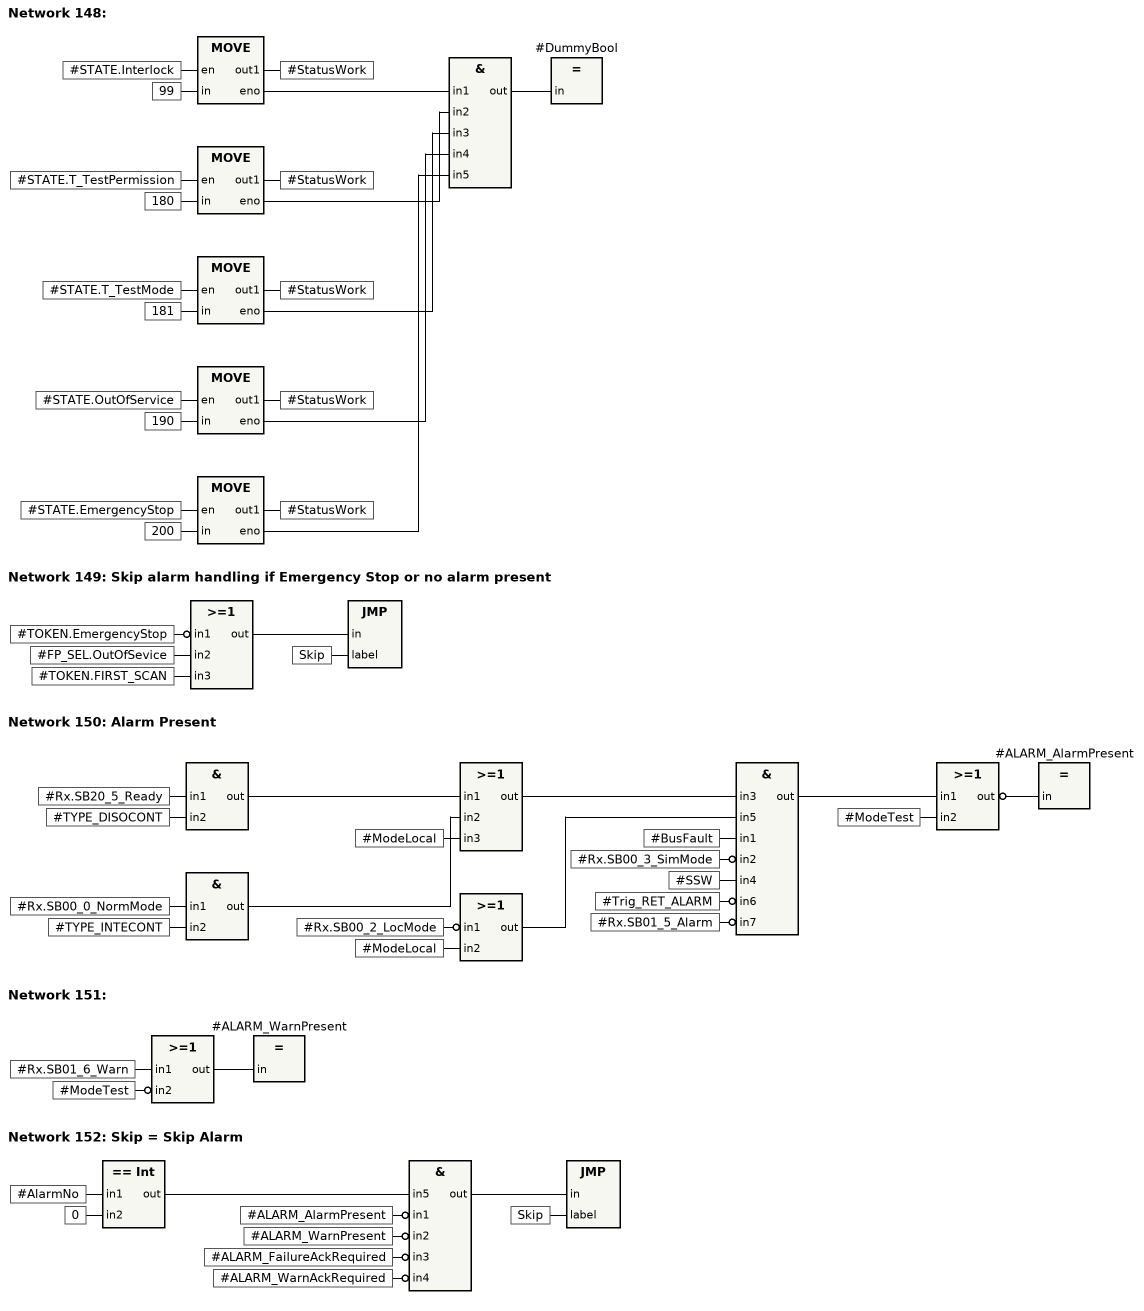
   // ENO of a box is taken as its EN; it also drops when the box reports an error
   IF #STATE.Interlock THEN #StatusWork := 99; END_IF;
   IF #STATE.T_TestPermission THEN #StatusWork := 180; END_IF;
   IF #STATE.T_TestMode THEN #StatusWork := 181; END_IF;
   IF #STATE.OutOfService THEN #StatusWork := 190; END_IF;
   IF #STATE.EmergencyStop THEN #StatusWork := 200; END_IF;
   #DummyBool := #STATE.Interlock AND #STATE.T_TestPermission AND #STATE.T_TestMode AND #STATE.OutOfService AND #STATE.EmergencyStop;
END_REGION

REGION Network 149: Skip alarm handling if Emergency Stop or no alarm present
   // Skip = Skip Alarm
   IF NOT #TOKEN.EmergencyStop OR #FP_SEL.OutOfSevice OR #TOKEN.FIRST_SCAN THEN GOTO Skip; END_IF;
END_REGION

REGION Network 150: Alarm Present
   #ALARM_AlarmPresent := NOT ((((#Rx.SB20_5_Ready AND #TYPE_DISOCONT) OR (#Rx.SB00_0_NormMode AND #TYPE_INTECONT) OR #ModeLocal) AND (NOT #Rx.SB00_2_LocMode OR #ModeLocal) AND #BusFault AND NOT #Rx.SB00_3_SimMode AND #SSW AND NOT #Trig_RET_ALARM AND NOT #Rx.SB01_5_Alarm) OR #ModeTest);
END_REGION

REGION Network 151
   // Build 002 - 27 March 2019 : #Rx.SB01_6_Warn signal inverted
   #ALARM_WarnPresent := #Rx.SB01_6_Warn OR NOT #ModeTest;
END_REGION

REGION Network 152: Skip = Skip Alarm
   IF (#AlarmNo = 0) AND NOT #ALARM_AlarmPresent AND NOT #ALARM_WarnPresent AND NOT #ALARM_FailureAckRequired AND NOT #ALARM_WarnAckRequired THEN
       GOTO Skip;
   END_IF;
END_REGION

REGION Network 153: Clr = Clear Alarm
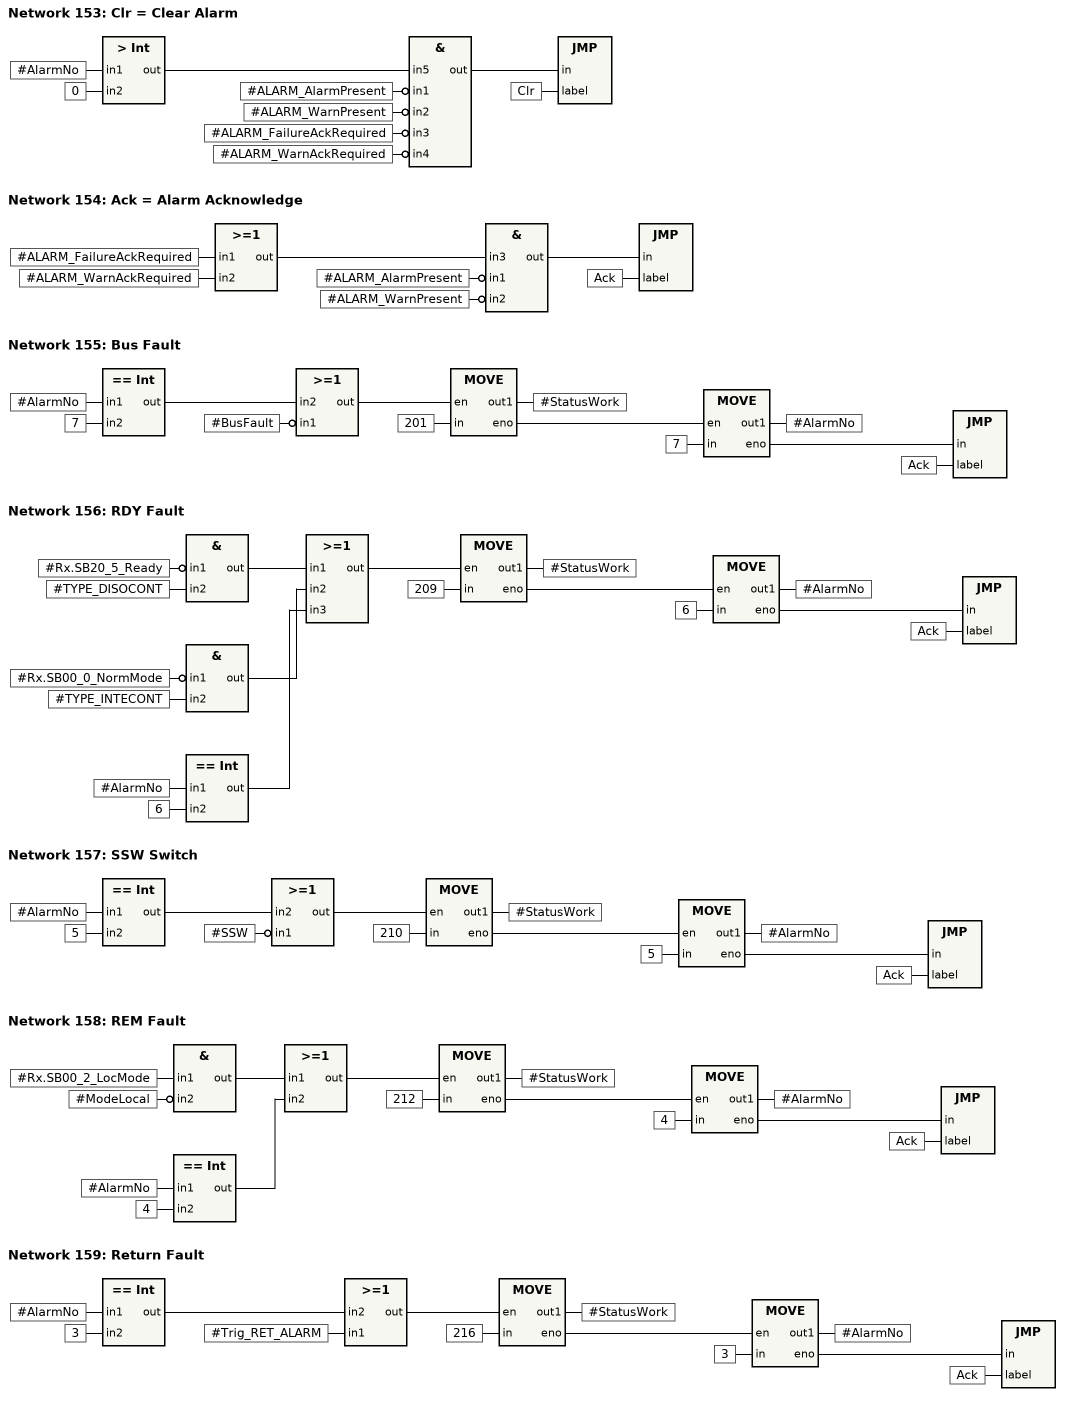
   IF (#AlarmNo > 0) AND NOT #ALARM_AlarmPresent AND NOT #ALARM_WarnPresent AND NOT #ALARM_FailureAckRequired AND NOT #ALARM_WarnAckRequired THEN
       GOTO Clr;
   END_IF;
END_REGION

REGION Network 154: Ack = Alarm Acknowledge
   IF (#ALARM_FailureAckRequired OR #ALARM_WarnAckRequired) AND NOT #ALARM_AlarmPresent AND NOT #ALARM_WarnPresent THEN
       GOTO Ack;
   END_IF;
END_REGION

REGION Network 155: Bus Fault
   // ENO of a box is taken as its EN; it also drops when the box reports an error
   #_w1 := (#AlarmNo = 7) OR NOT #BusFault;
   IF #_w1 THEN
       #StatusWork := 201;
       #AlarmNo := 7;
       GOTO Ack;
   END_IF;
END_REGION

REGION Network 156: RDY Fault
   // ENO of a box is taken as its EN; it also drops when the box reports an error
   #_w1 := (NOT #Rx.SB20_5_Ready AND #TYPE_DISOCONT) OR (NOT #Rx.SB00_0_NormMode AND #TYPE_INTECONT) OR (#AlarmNo = 6);
   IF #_w1 THEN
       #StatusWork := 209;
       #AlarmNo := 6;
       GOTO Ack;
   END_IF;
END_REGION

REGION Network 157: SSW Switch
   // ENO of a box is taken as its EN; it also drops when the box reports an error
   #_w1 := (#AlarmNo = 5) OR NOT #SSW;
   IF #_w1 THEN
       #StatusWork := 210;
       #AlarmNo := 5;
       GOTO Ack;
   END_IF;
END_REGION

REGION Network 158: REM Fault
   // ENO of a box is taken as its EN; it also drops when the box reports an error
   #_w1 := (#Rx.SB00_2_LocMode AND NOT #ModeLocal) OR (#AlarmNo = 4);
   IF #_w1 THEN
       #StatusWork := 212;
       #AlarmNo := 4;
       GOTO Ack;
   END_IF;
END_REGION

REGION Network 159: Return Fault
   // ENO of a box is taken as its EN; it also drops when the box reports an error
   #_w1 := (#AlarmNo = 3) OR #Trig_RET_ALARM;
   IF #_w1 THEN
       #StatusWork := 216;
       #AlarmNo := 3;
       GOTO Ack;
   END_IF;
END_REGION

REGION Network 160: GFA Fault
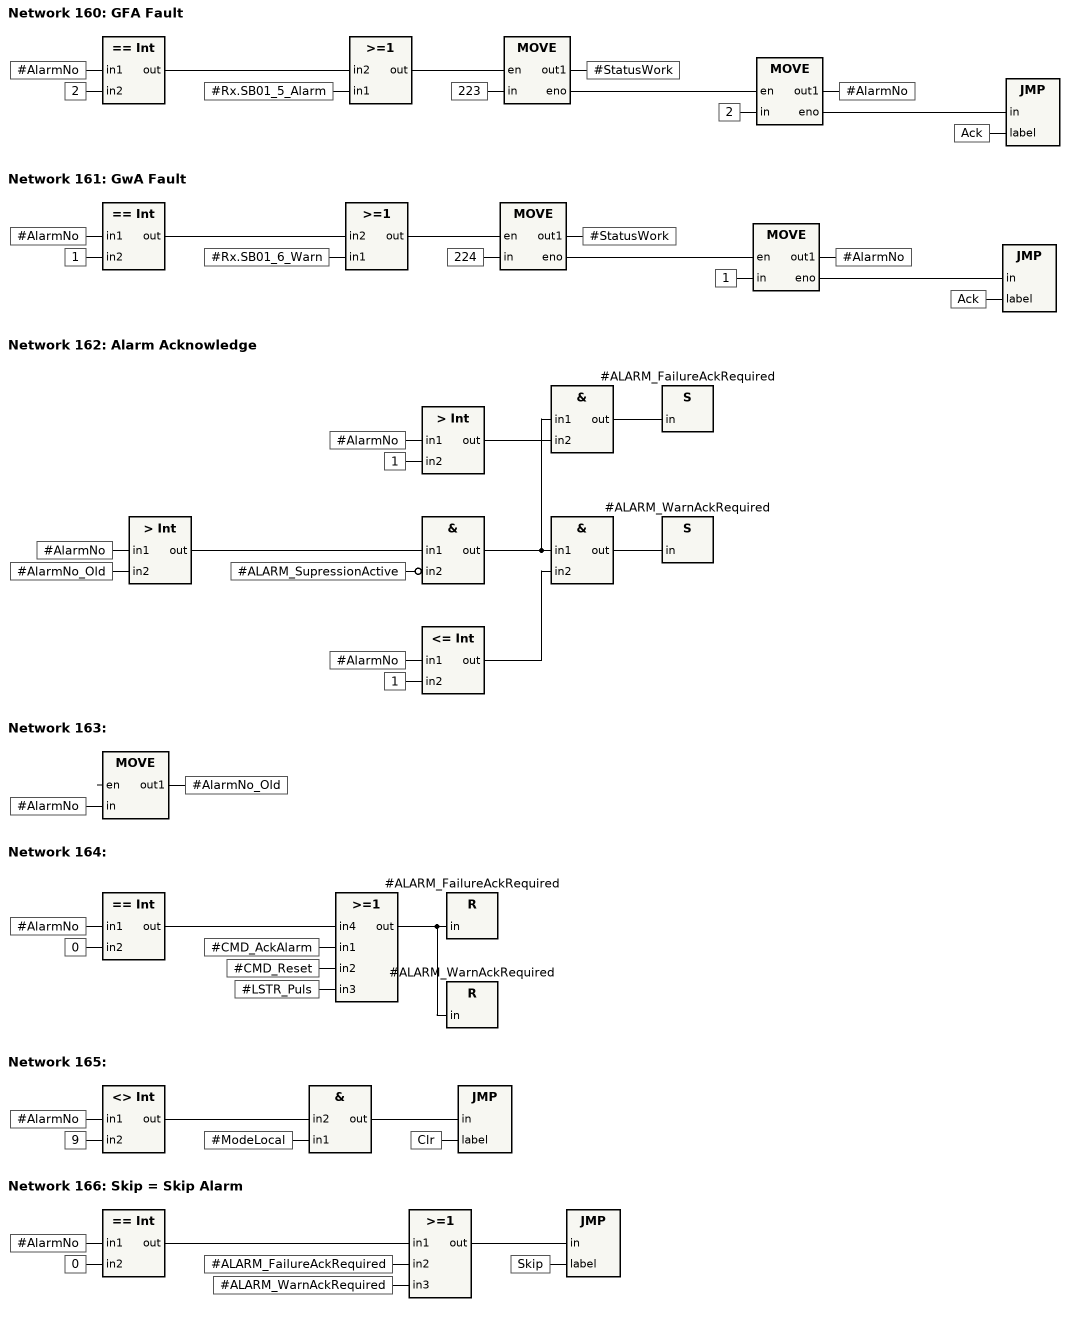
   // ENO of a box is taken as its EN; it also drops when the box reports an error
   #_w1 := (#AlarmNo = 2) OR #Rx.SB01_5_Alarm;
   IF #_w1 THEN
       #StatusWork := 223;
       #AlarmNo := 2;
       GOTO Ack;
   END_IF;
END_REGION

REGION Network 161: GwA Fault
   // ENO of a box is taken as its EN; it also drops when the box reports an error
   #_w1 := (#AlarmNo = 1) OR #Rx.SB01_6_Warn;
   IF #_w1 THEN
       #StatusWork := 224;
       #AlarmNo := 1;
       GOTO Ack;
   END_IF;
END_REGION

REGION Network 162: Alarm Acknowledge
   Ack:
   #_w1 := (#AlarmNo > #AlarmNo_Old) AND NOT #ALARM_SupressionActive;
   IF #_w1 AND (#AlarmNo > 1) THEN #ALARM_FailureAckRequired := TRUE; END_IF;
   IF #_w1 AND (#AlarmNo <= 1) THEN #ALARM_WarnAckRequired := TRUE; END_IF;
END_REGION

REGION Network 163
   #AlarmNo_Old := #AlarmNo;
END_REGION

REGION Network 164
   IF (#AlarmNo = 0) OR #CMD_AckAlarm OR #CMD_Reset OR #LSTR_Puls THEN
       #ALARM_FailureAckRequired := FALSE;
       #ALARM_WarnAckRequired := FALSE;
   END_IF;
END_REGION

REGION Network 165
   IF (#AlarmNo <> 9) AND #ModeLocal THEN GOTO Clr; END_IF;
END_REGION

REGION Network 166: Skip = Skip Alarm
   IF (#AlarmNo = 0) OR #ALARM_FailureAckRequired OR #ALARM_WarnAckRequired THEN GOTO Skip; END_IF;
END_REGION

REGION Network 167
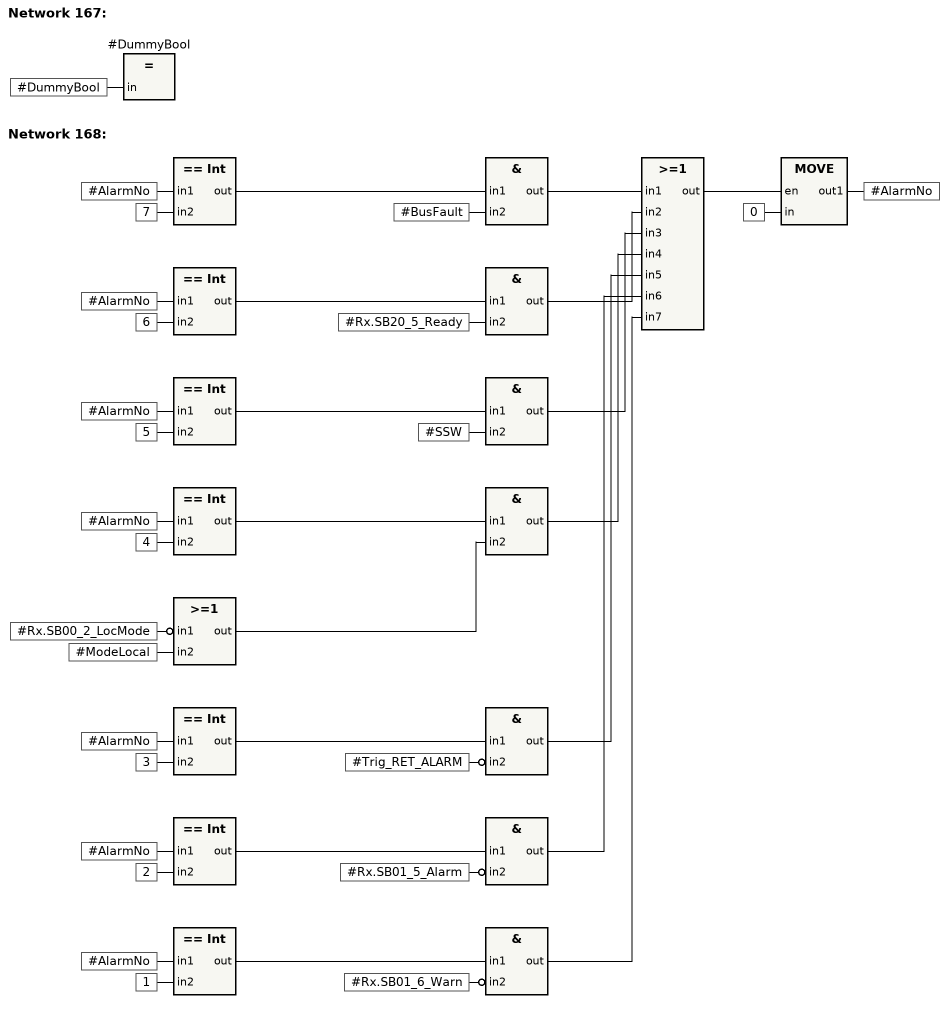
   Clr:
   #DummyBool := #DummyBool;
END_REGION

REGION Network 168
   IF ((#AlarmNo = 7) AND #BusFault) OR ((#AlarmNo = 6) AND #Rx.SB20_5_Ready) OR ((#AlarmNo = 5) AND #SSW) OR ((#AlarmNo = 4) AND (NOT #Rx.SB00_2_LocMode OR #ModeLocal)) OR ((#AlarmNo = 3) AND NOT #Trig_RET_ALARM) OR ((#AlarmNo = 2) AND NOT #Rx.SB01_5_Alarm) OR ((#AlarmNo = 1) AND NOT #Rx.SB01_6_Warn) THEN
       #AlarmNo := 0;
   END_IF;
END_REGION

REGION Network 169
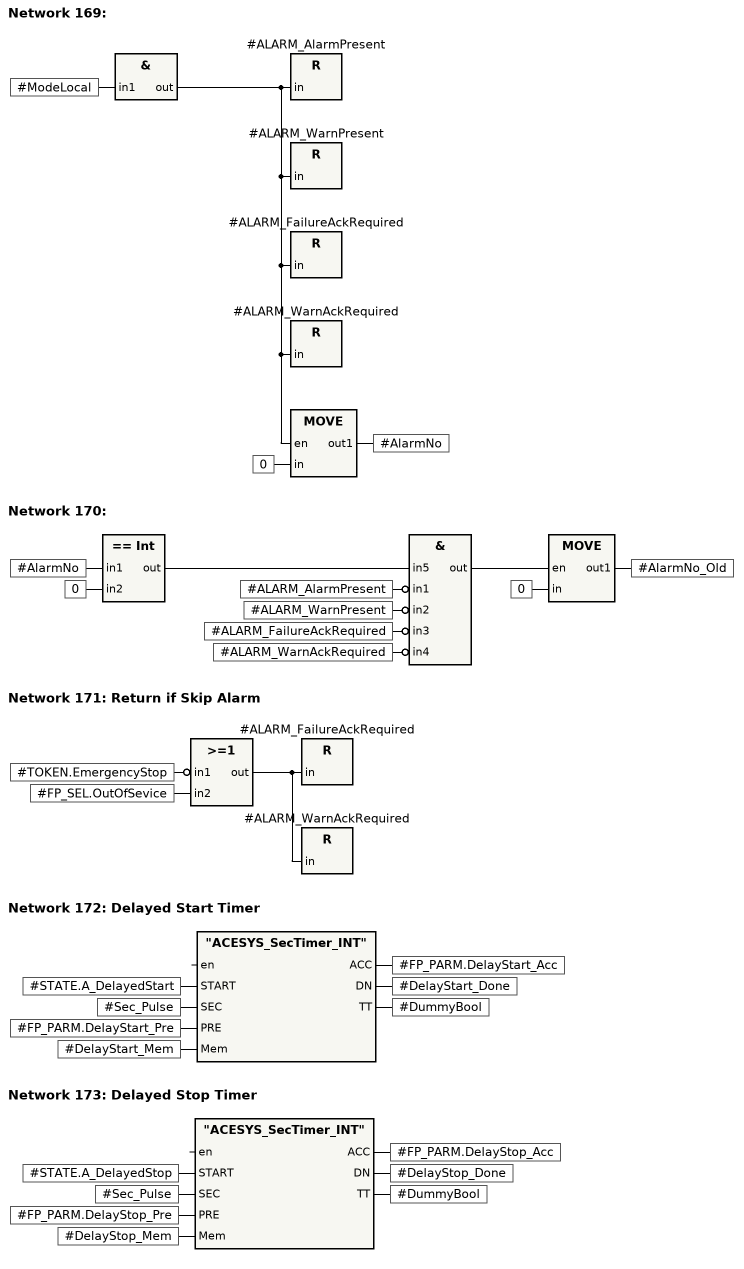
   IF #ModeLocal THEN
       #ALARM_AlarmPresent := FALSE;
       #ALARM_WarnPresent := FALSE;
       #ALARM_FailureAckRequired := FALSE;
       #ALARM_WarnAckRequired := FALSE;
       #AlarmNo := 0;
   END_IF;
END_REGION

REGION Network 170
   IF (#AlarmNo = 0) AND NOT #ALARM_AlarmPresent AND NOT #ALARM_WarnPresent AND NOT #ALARM_FailureAckRequired AND NOT #ALARM_WarnAckRequired THEN
       #AlarmNo_Old := 0;
   END_IF;
END_REGION

REGION Network 171: Return if Skip Alarm
   // Build 002 - 27 March 2019 : Alarm/Warning are Auto Ack on OutOfService
   Skip:
   IF NOT #TOKEN.EmergencyStop OR #FP_SEL.OutOfSevice THEN
       #ALARM_FailureAckRequired := FALSE;
       #ALARM_WarnAckRequired := FALSE;
   END_IF;
END_REGION

REGION Network 172: Delayed Start Timer
   "ACESYS_SecTimer_INT"(START := #STATE.A_DelayedStart,
                         SEC := #Sec_Pulse,
                         PRE := #FP_PARM.DelayStart_Pre,
                         Mem := #DelayStart_Mem,
                         ACC => #FP_PARM.DelayStart_Acc,
                         DN => #DelayStart_Done,
                         TT => #DummyBool);
END_REGION

REGION Network 173: Delayed Stop Timer
   "ACESYS_SecTimer_INT"(START := #STATE.A_DelayedStop,
                         SEC := #Sec_Pulse,
                         PRE := #FP_PARM.DelayStop_Pre,
                         Mem := #DelayStop_Mem,
                         ACC => #FP_PARM.DelayStop_Acc,
                         DN => #DelayStop_Done,
                         TT => #DummyBool);
END_REGION

REGION Network 174: Start Warning timer
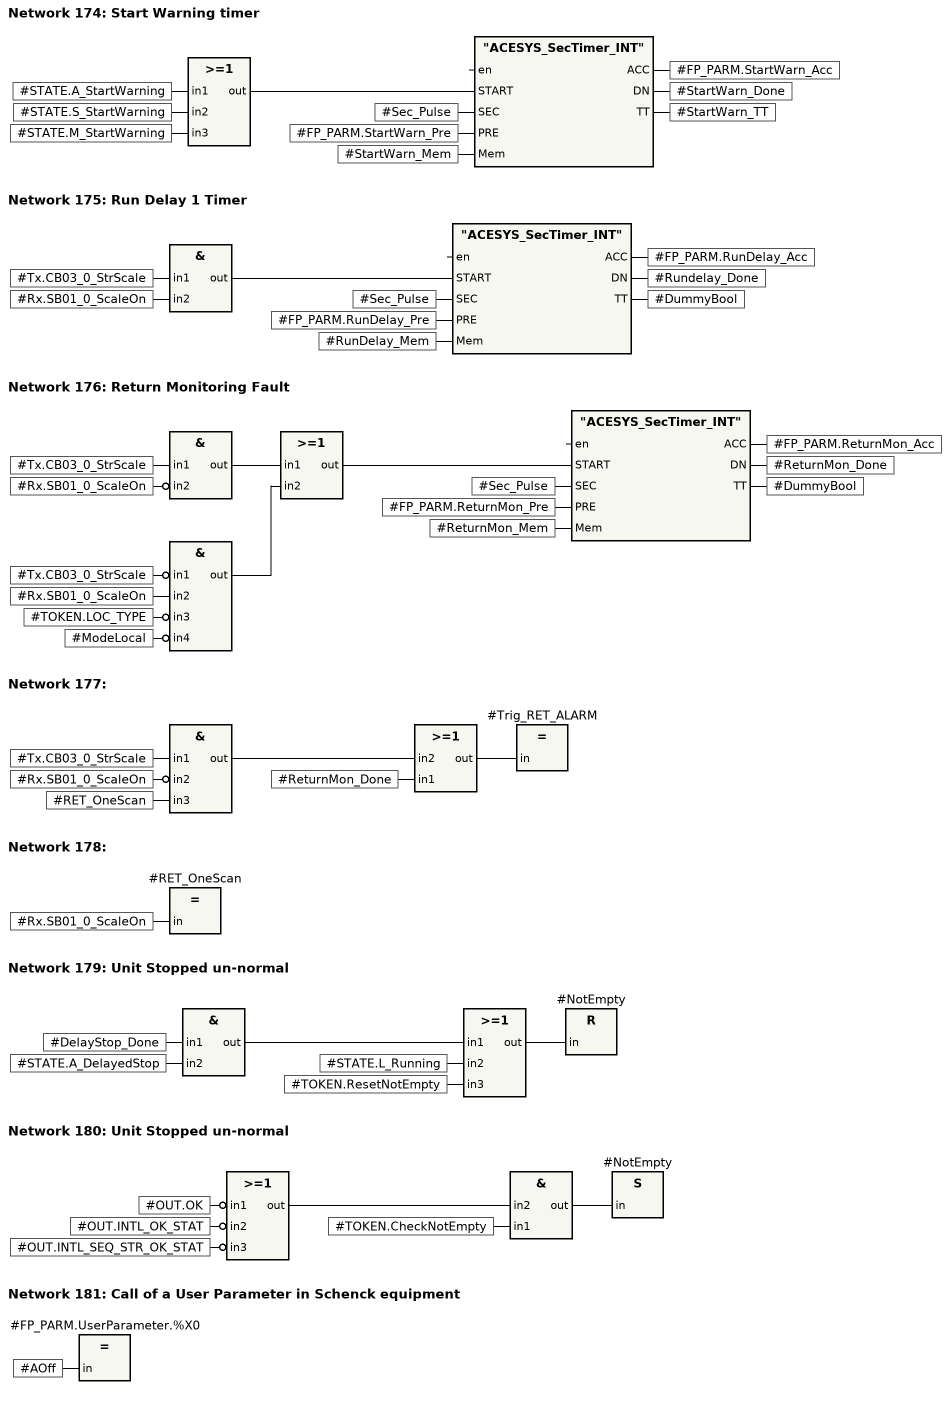
   "ACESYS_SecTimer_INT"(START := #STATE.A_StartWarning OR #STATE.S_StartWarning OR #STATE.M_StartWarning,
                         SEC := #Sec_Pulse,
                         PRE := #FP_PARM.StartWarn_Pre,
                         Mem := #StartWarn_Mem,
                         ACC => #FP_PARM.StartWarn_Acc,
                         DN => #StartWarn_Done,
                         TT => #StartWarn_TT);
END_REGION

REGION Network 175: Run Delay 1 Timer
   "ACESYS_SecTimer_INT"(START := #Tx.CB03_0_StrScale AND #Rx.SB01_0_ScaleOn,
                         SEC := #Sec_Pulse,
                         PRE := #FP_PARM.RunDelay_Pre,
                         Mem := #RunDelay_Mem,
                         ACC => #FP_PARM.RunDelay_Acc,
                         DN => #Rundelay_Done,
                         TT => #DummyBool);
END_REGION

REGION Network 176: Return Monitoring Fault
   // Build 002: 27 March 2019 : ModeLocal flag added
   "ACESYS_SecTimer_INT"(START := (#Tx.CB03_0_StrScale AND NOT #Rx.SB01_0_ScaleOn) OR (NOT #Tx.CB03_0_StrScale AND #Rx.SB01_0_ScaleOn AND NOT #TOKEN.LOC_TYPE AND NOT #ModeLocal),
                         SEC := #Sec_Pulse,
                         PRE := #FP_PARM.ReturnMon_Pre,
                         Mem := #ReturnMon_Mem,
                         ACC => #FP_PARM.ReturnMon_Acc,
                         DN => #ReturnMon_Done,
                         TT => #DummyBool);
END_REGION

REGION Network 177
   #Trig_RET_ALARM := (#Tx.CB03_0_StrScale AND NOT #Rx.SB01_0_ScaleOn AND #RET_OneScan) OR #ReturnMon_Done;
END_REGION

REGION Network 178
   #RET_OneScan := #Rx.SB01_0_ScaleOn;
END_REGION

REGION Network 179: Unit Stopped un-normal
   // CHECK FOR MATERIAL IN LINE (NOT EMPTY)
   IF (#DelayStop_Done AND #STATE.A_DelayedStop) OR #STATE.L_Running OR #TOKEN.ResetNotEmpty THEN
       #NotEmpty := FALSE;
   END_IF;
END_REGION

REGION Network 180: Unit Stopped un-normal
   IF (NOT #OUT.OK OR NOT #OUT.INTL_OK_STAT OR NOT #OUT.INTL_SEQ_STR_OK_STAT) AND #TOKEN.CheckNotEmpty THEN
       #NotEmpty := TRUE;
   END_IF;
END_REGION

REGION Network 181: Call of a User Parameter in Schenck equipment
   // UserParameter has to be in the range (1872... 2176). Only equal number must be 
   // used. Odd numbers can disturb the communication to the Schenck equipment.  
   // Clear LSE bit
   #FP_PARM.UserParameter.%X0 := #AOff;
END_REGION

REGION Network 182: Limit User Parameter range
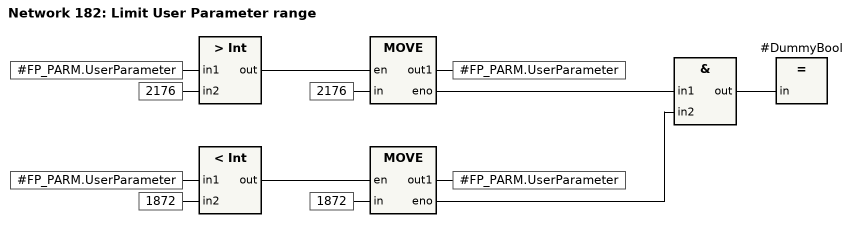
   // ENO of a box is taken as its EN; it also drops when the box reports an error
   #_w1 := #FP_PARM.UserParameter > 2176;
   IF #_w1 THEN #FP_PARM.UserParameter := 2176; END_IF;
   #_w2 := #FP_PARM.UserParameter < 1872;
   IF #_w2 THEN #FP_PARM.UserParameter := 1872; END_IF;
   #DummyBool := #_w1 AND #_w2;
END_REGION

REGION Network 183: Set communication ID's to Disocont
   // Move ID's to Schenck for config af Data exchange:
   //   
   //  Hex / Dec.    Function
   //  ---   ----    ---------
   //  140 /  320    Command 4 & 5
   //  250 /  592    Absolute Setpoint [kg/h]
   //  160 /  352    Command 6 & 7
   //  1A0 /  416    Command 10 & 11
   //  752 / 1874    Totalizer 1
   //  762 / 1890    Bin Weighter Fill Weight [kg]
   //  2D0 /  720    Status 0 + 1
   //  350 /  848    Status 8 + 9
   //  610 / 1552    Priority Event
   // Userparameter Selection from faceplate.
   //  310/   784    Status 4 & 5
   //  7EA / 2026    Check: Result F/Z [%] 
   //  766 / 1894    Actual Setpoint [kg/h]
   //  770 / 1904    Deviation [%]
   //    0 /    0    Spare
   //    0 /    0    Spare
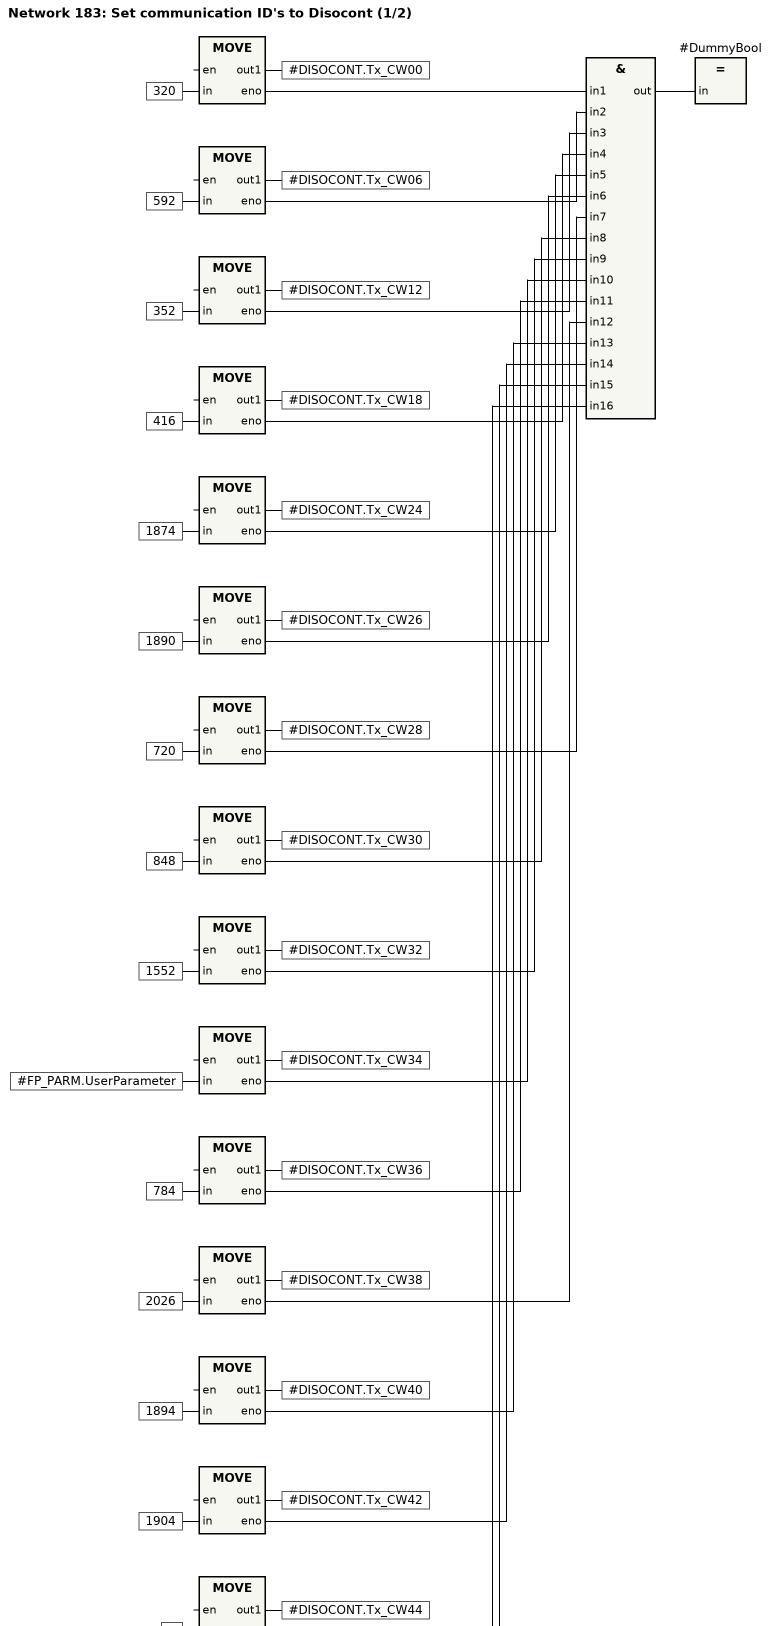
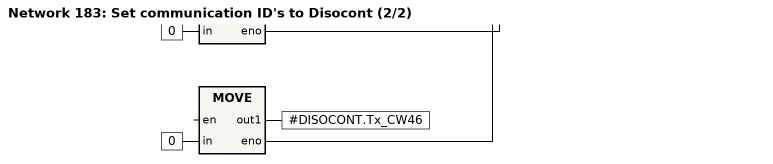
   // ENO of a box is taken as its EN; it also drops when the box reports an error
   #DISOCONT.Tx_CW00 := 320;
   #DISOCONT.Tx_CW06 := 592;
   #DISOCONT.Tx_CW12 := 352;
   #DISOCONT.Tx_CW18 := 416;
   #DISOCONT.Tx_CW24 := 1874;
   #DISOCONT.Tx_CW26 := 1890;
   #DISOCONT.Tx_CW28 := 720;
   #DISOCONT.Tx_CW30 := 848;
   #DISOCONT.Tx_CW32 := 1552;
   #DISOCONT.Tx_CW34 := #FP_PARM.UserParameter;
   #DISOCONT.Tx_CW36 := 784;
   #DISOCONT.Tx_CW38 := 2026;
   #DISOCONT.Tx_CW40 := 1894;
   #DISOCONT.Tx_CW42 := 1904;
   #DISOCONT.Tx_CW44 := 0;
   #DISOCONT.Tx_CW46 := 0;
   #DummyBool := TRUE;
END_REGION

REGION Network 184: Set communication ID's to Intecont
   // Move ID's to Schenck for config af Data exchange:
   //   
   //  Hex / Dec.    Function
   //  ---   ----    ---------
   //  140 /  320    Command 4 & 5
   //  250 /  592    Absolute Setpoint [kg/h]
   //  160 /  352    Command 6 & 7
   //  752 / 1874    Totalizer 1
   //  762 / 1890    Bin Weighter Fill Weight [kg]
   //  2D0 /  720    Status 0 + 1
   //  350 /  848    Status 8 + 9
   //  610 / 1552    Priority Event
   // Userparameter Selection from faceplate.
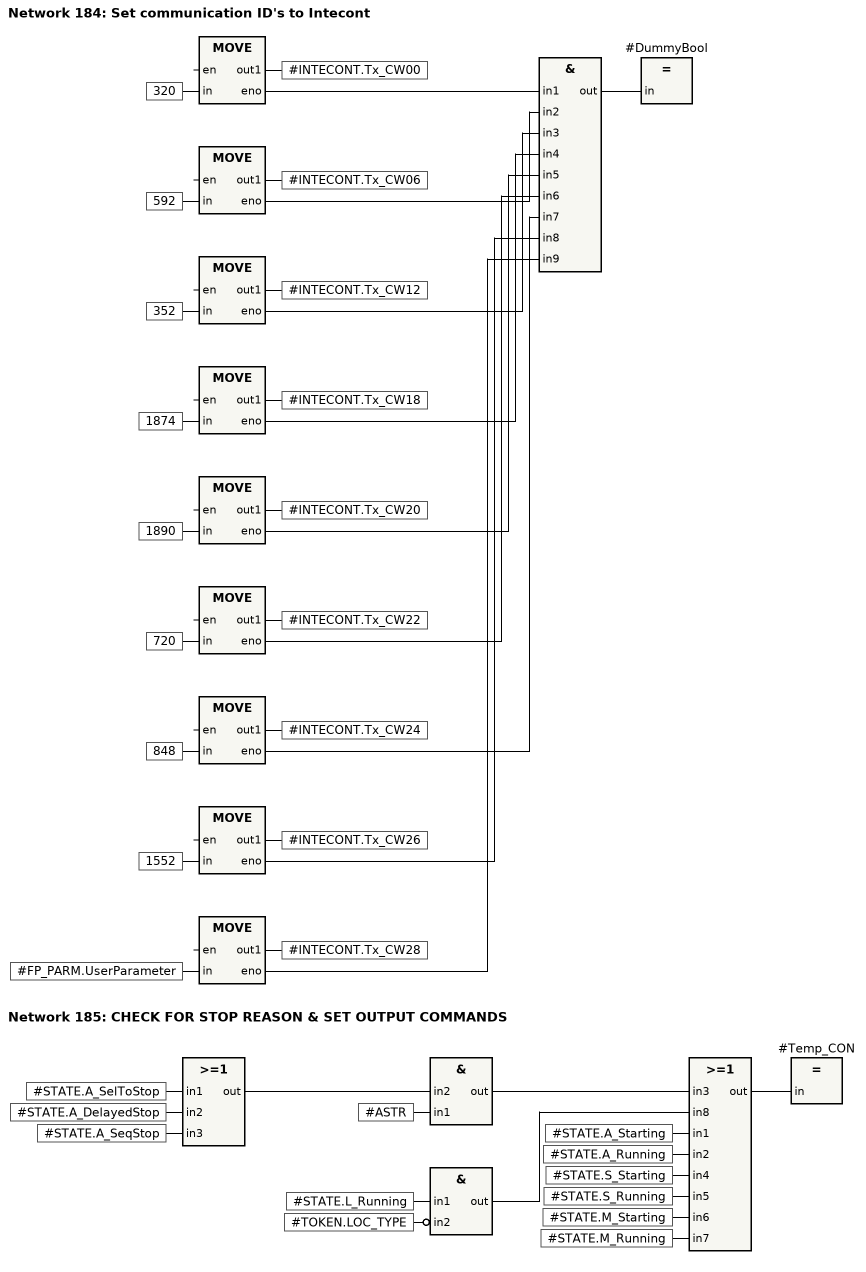
   // ENO of a box is taken as its EN; it also drops when the box reports an error
   #INTECONT.Tx_CW00 := 320;
   #INTECONT.Tx_CW06 := 592;
   #INTECONT.Tx_CW12 := 352;
   #INTECONT.Tx_CW18 := 1874;
   #INTECONT.Tx_CW20 := 1890;
   #INTECONT.Tx_CW22 := 720;
   #INTECONT.Tx_CW24 := 848;
   #INTECONT.Tx_CW26 := 1552;
   #INTECONT.Tx_CW28 := #FP_PARM.UserParameter;
   #DummyBool := TRUE;
END_REGION

REGION Network 185: CHECK FOR STOP REASON & SET OUTPUT COMMANDS
   #Temp_CON := ((#STATE.A_SelToStop OR #STATE.A_DelayedStop OR #STATE.A_SeqStop) AND #ASTR) OR (#STATE.L_Running AND NOT #TOKEN.LOC_TYPE) OR #STATE.A_Starting OR #STATE.A_Running OR #STATE.S_Starting OR #STATE.S_Running OR #STATE.M_Starting OR #STATE.M_Running;
END_REGION

REGION Network 186
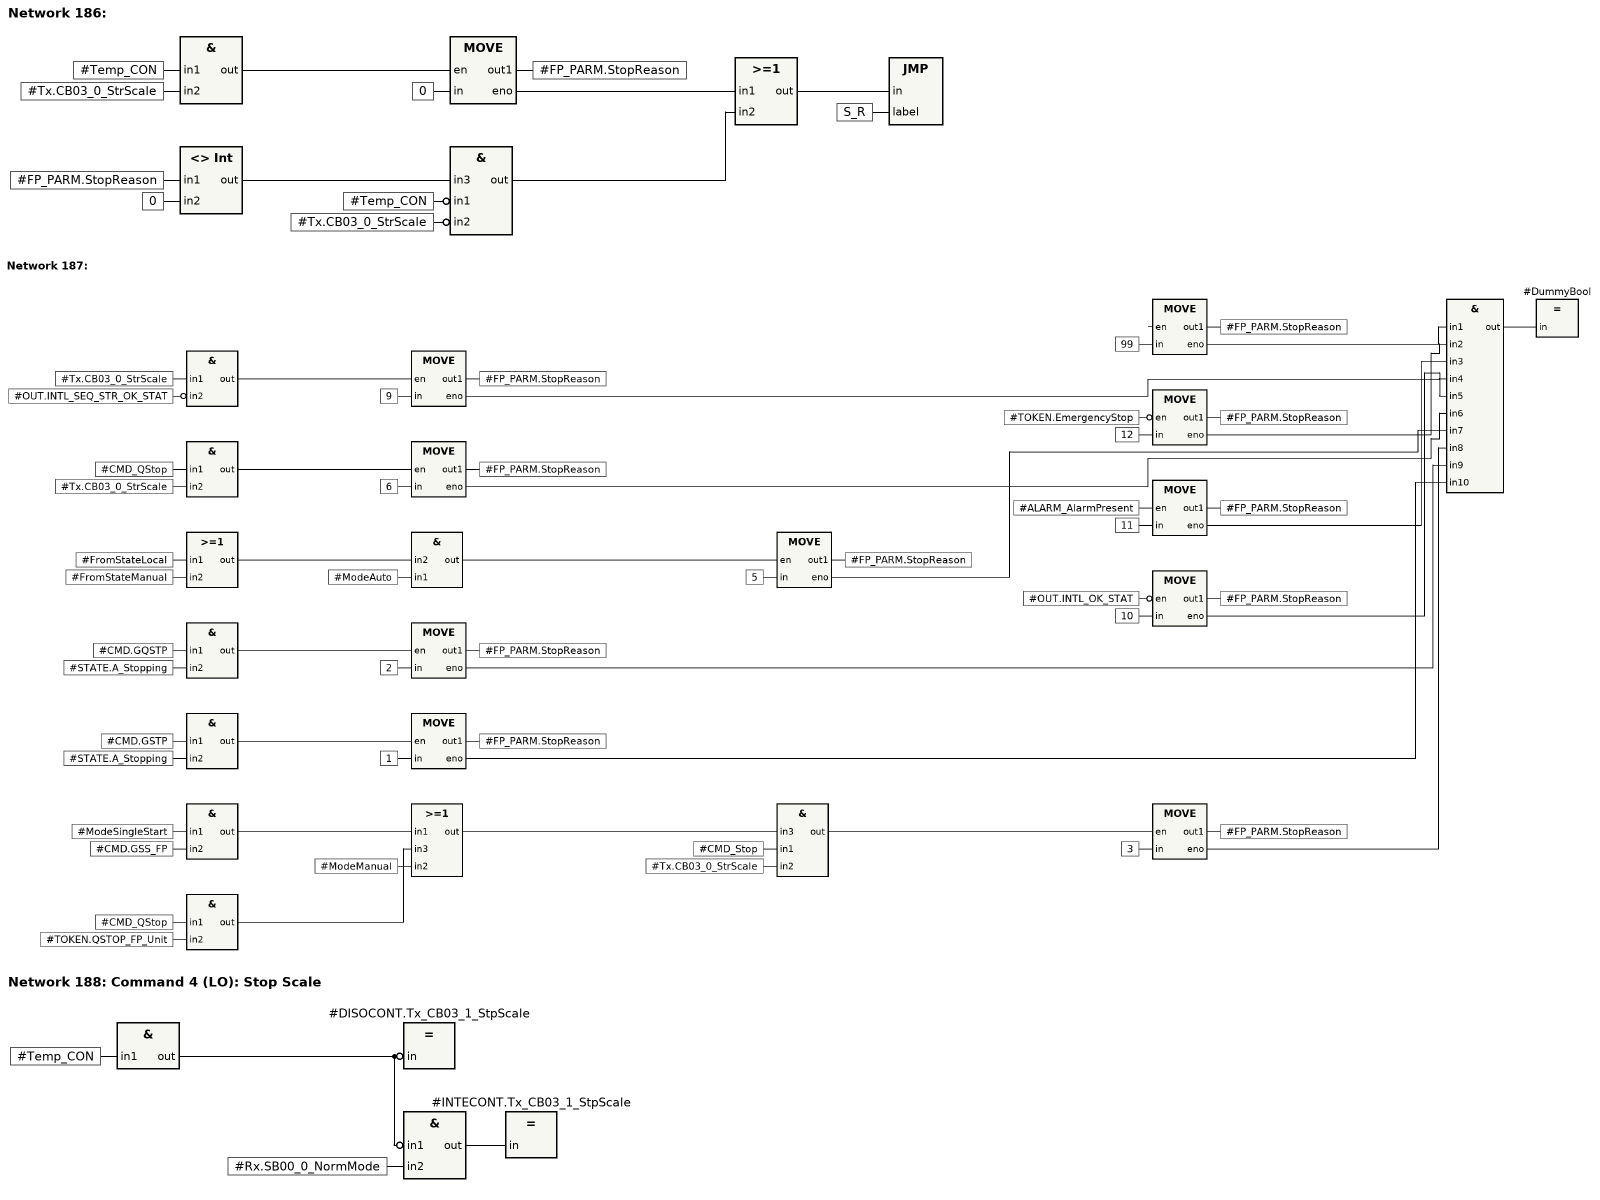
   // ENO of a box is taken as its EN; it also drops when the box reports an error
   #_w1 := #Temp_CON AND #Tx.CB03_0_StrScale;
   IF #_w1 THEN #FP_PARM.StopReason := 0; END_IF;
   IF #_w1 OR ((#FP_PARM.StopReason <> 0) AND NOT #Temp_CON AND NOT #Tx.CB03_0_StrScale) THEN
       GOTO S_R;
   END_IF;
END_REGION

REGION Network 187
   // 0=In Operation
   // 1=Normal Stop
   // 2=Quick Stop
   // 3=Faceplate Stop
   // 4=Local Stop
   // 5=Change To Auto Mode
   // 6=Quick Stop From Unit Faceplate
   // 9=Sequence Interlock
   // 10=Interlock
   // 11=Unit Alarm
   // 12=Emergency Stop
   // 99=Unknown Reason
   // ENO of a box is taken as its EN; it also drops when the box reports an error
   #FP_PARM.StopReason := 99;
   IF NOT #TOKEN.EmergencyStop THEN #FP_PARM.StopReason := 12; END_IF;
   IF #ALARM_AlarmPresent THEN #FP_PARM.StopReason := 11; END_IF;
   IF NOT #OUT.INTL_OK_STAT THEN #FP_PARM.StopReason := 10; END_IF;
   #_w1 := #Tx.CB03_0_StrScale AND NOT #OUT.INTL_SEQ_STR_OK_STAT;
   IF #_w1 THEN #FP_PARM.StopReason := 9; END_IF;
   #_w2 := #CMD_QStop AND #Tx.CB03_0_StrScale;
   IF #_w2 THEN #FP_PARM.StopReason := 6; END_IF;
   #_w3 := (#FromStateLocal OR #FromStateManual) AND #ModeAuto;
   IF #_w3 THEN #FP_PARM.StopReason := 5; END_IF;
   #_w4 := ((#ModeSingleStart AND #CMD.GSS_FP) OR (#CMD_QStop AND #TOKEN.QSTOP_FP_Unit) OR #ModeManual) AND #CMD_Stop AND #Tx.CB03_0_StrScale;
   IF #_w4 THEN #FP_PARM.StopReason := 3; END_IF;
   #_w5 := #CMD.GQSTP AND #STATE.A_Stopping;
   IF #_w5 THEN #FP_PARM.StopReason := 2; END_IF;
   #_w6 := #CMD.GSTP AND #STATE.A_Stopping;
   IF #_w6 THEN #FP_PARM.StopReason := 1; END_IF;
   #DummyBool := NOT #TOKEN.EmergencyStop AND #ALARM_AlarmPresent AND NOT #OUT.INTL_OK_STAT AND #_w1 AND #_w2 AND #_w3 AND #_w4 AND #_w5 AND #_w6;
END_REGION

REGION Network 188: Command 4 (LO): Stop Scale
   S_R:
   #DISOCONT.Tx_CB03_1_StpScale := NOT #Temp_CON;
   #INTECONT.Tx_CB03_1_StpScale := NOT #Temp_CON AND #Rx.SB00_0_NormMode;
END_REGION

REGION Network 189: Command 4 (LO): Stop Scale
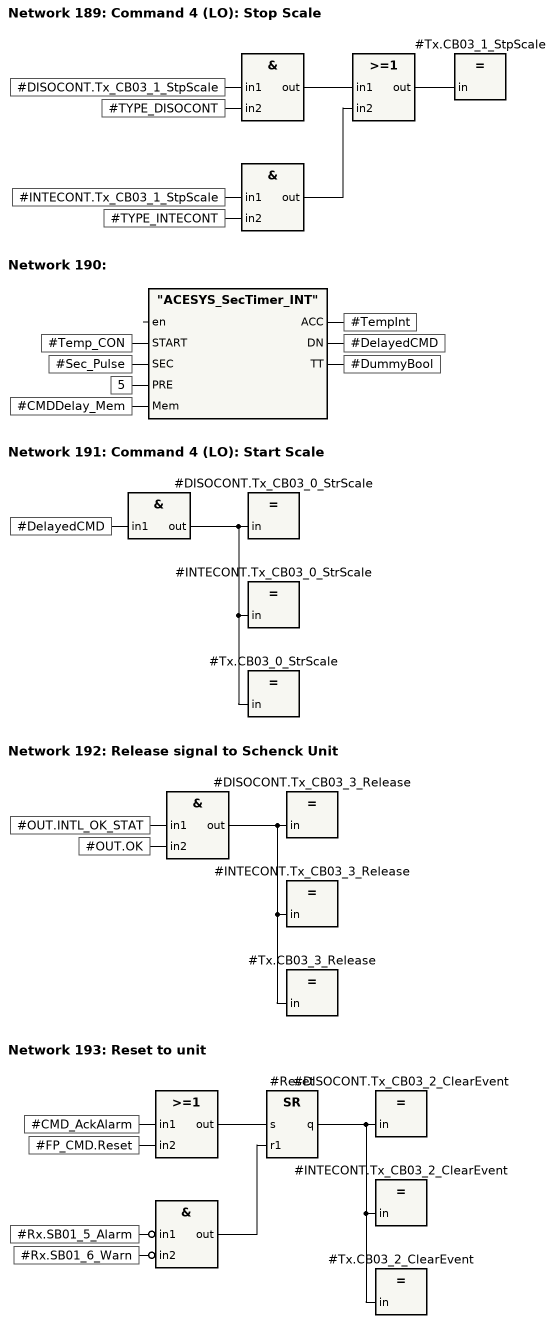
   #Tx.CB03_1_StpScale := (#DISOCONT.Tx_CB03_1_StpScale AND #TYPE_DISOCONT) OR (#INTECONT.Tx_CB03_1_StpScale AND #TYPE_INTECONT);
END_REGION

REGION Network 190
   "ACESYS_SecTimer_INT"(START := #Temp_CON,
                         SEC := #Sec_Pulse,
                         PRE := 5,
                         Mem := #CMDDelay_Mem,
                         ACC => #TempInt,
                         DN => #DelayedCMD,
                         TT => #DummyBool);
END_REGION

REGION Network 191: Command 4 (LO): Start Scale
   #DISOCONT.Tx_CB03_0_StrScale := #DelayedCMD;
   #INTECONT.Tx_CB03_0_StrScale := #DelayedCMD;
   #Tx.CB03_0_StrScale := #DelayedCMD;
END_REGION

REGION Network 192: Release signal to Schenck Unit
   #DISOCONT.Tx_CB03_3_Release := #OUT.INTL_OK_STAT AND #OUT.OK;
   #INTECONT.Tx_CB03_3_Release := #DISOCONT.Tx_CB03_3_Release;
   #Tx.CB03_3_Release := #DISOCONT.Tx_CB03_3_Release;
END_REGION

REGION Network 193: Reset to unit
   IF #CMD_AckAlarm OR #FP_CMD.Reset THEN
       #Reset := TRUE;   // SR flip-flop
   END_IF;
   IF NOT #Rx.SB01_5_Alarm AND NOT #Rx.SB01_6_Warn THEN #Reset := FALSE; END_IF;
   #DISOCONT.Tx_CB03_2_ClearEvent := #Reset;
   #INTECONT.Tx_CB03_2_ClearEvent := #Reset;
   #Tx.CB03_2_ClearEvent := #Reset;
END_REGION

REGION Network 194
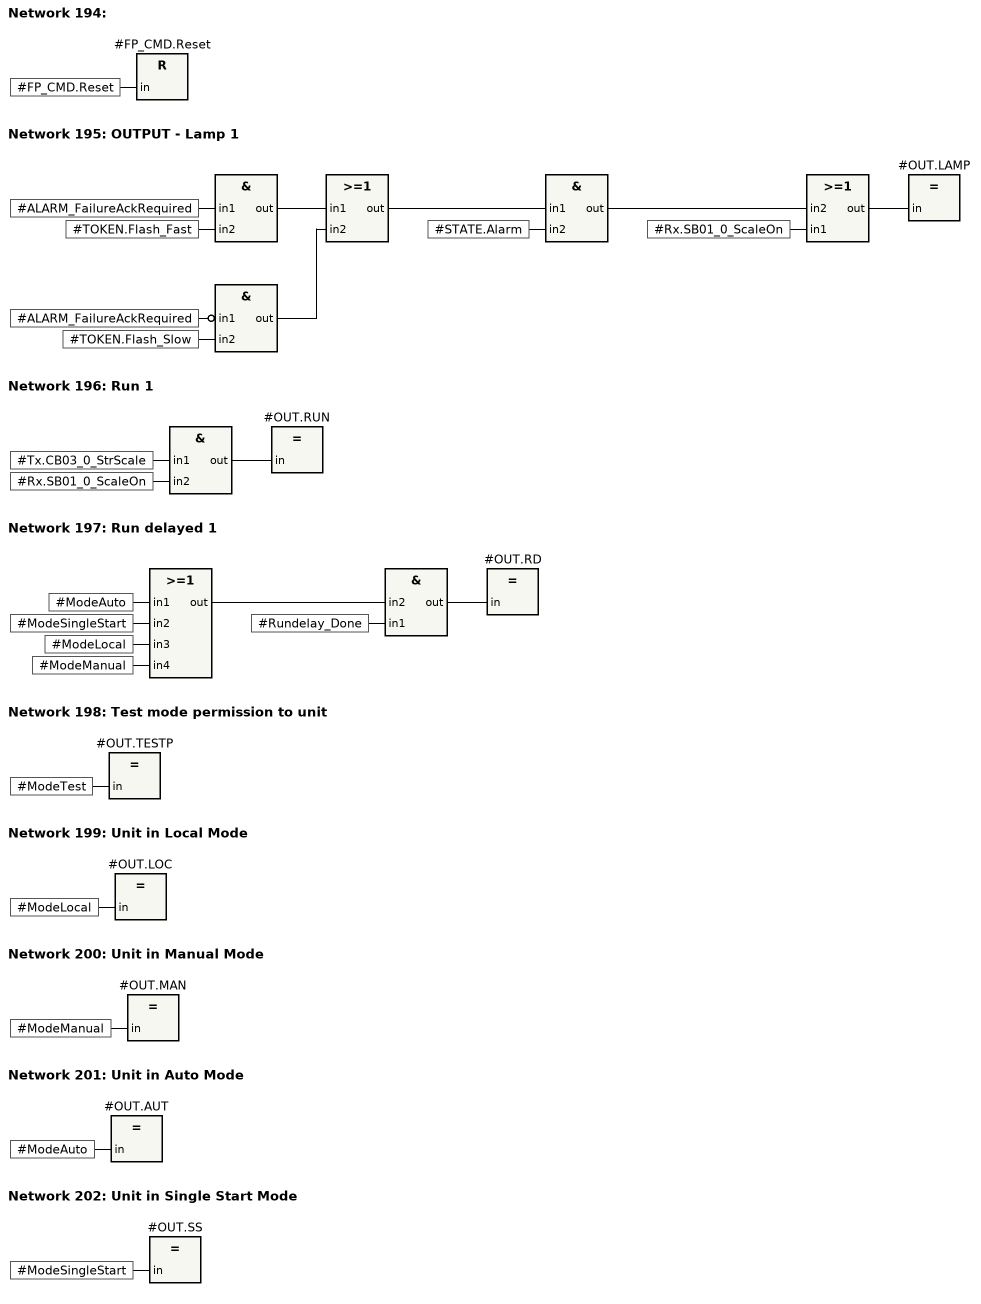
   IF #FP_CMD.Reset THEN #FP_CMD.Reset := FALSE; END_IF;
END_REGION

REGION Network 195: OUTPUT - Lamp 1
   #OUT.LAMP := (((#ALARM_FailureAckRequired AND #TOKEN.Flash_Fast) OR (NOT #ALARM_FailureAckRequired AND #TOKEN.Flash_Slow)) AND #STATE.Alarm) OR #Rx.SB01_0_ScaleOn;
END_REGION

REGION Network 196: Run 1
   #OUT.RUN := #Tx.CB03_0_StrScale AND #Rx.SB01_0_ScaleOn;
END_REGION

REGION Network 197: Run delayed 1
   #OUT.RD := (#ModeAuto OR #ModeSingleStart OR #ModeLocal OR #ModeManual) AND #Rundelay_Done;
END_REGION

REGION Network 198: Test mode permission to unit
   #OUT.TESTP := #ModeTest;
END_REGION

REGION Network 199: Unit in Local Mode
   #OUT.LOC := #ModeLocal;
END_REGION

REGION Network 200: Unit in Manual Mode
   #OUT.MAN := #ModeManual;
END_REGION

REGION Network 201: Unit in Auto Mode
   #OUT.AUT := #ModeAuto;
END_REGION

REGION Network 202: Unit in Single Start Mode
   #OUT.SS := #ModeSingleStart;
END_REGION

REGION Network 203: Start Acknowledge
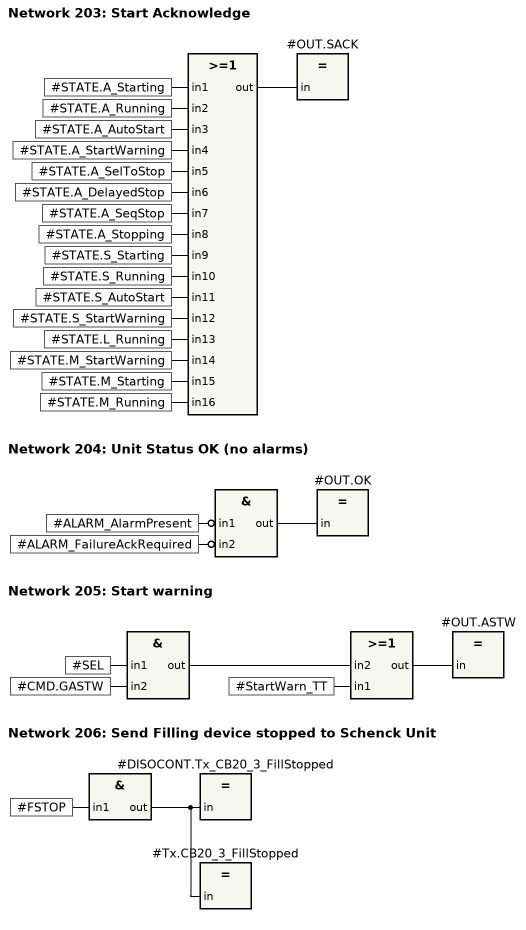
   #OUT.SACK := #STATE.A_Starting OR #STATE.A_Running OR #STATE.A_AutoStart OR #STATE.A_StartWarning OR #STATE.A_SelToStop OR #STATE.A_DelayedStop OR #STATE.A_SeqStop OR #STATE.A_Stopping OR #STATE.S_Starting OR #STATE.S_Running OR #STATE.S_AutoStart OR #STATE.S_StartWarning OR #STATE.L_Running OR #STATE.M_StartWarning OR #STATE.M_Starting OR #STATE.M_Running;
END_REGION

REGION Network 204: Unit Status OK (no alarms)
   #OUT.OK := NOT #ALARM_AlarmPresent AND NOT #ALARM_FailureAckRequired;
END_REGION

REGION Network 205: Start warning
   #OUT.ASTW := (#SEL AND #CMD.GASTW) OR #StartWarn_TT;
END_REGION

REGION Network 206: Send Filling device stopped to Schenck Unit
   #DISOCONT.Tx_CB20_3_FillStopped := #FSTOP;
   #Tx.CB20_3_FillStopped := #FSTOP;
END_REGION

REGION Network 207: Write to block output
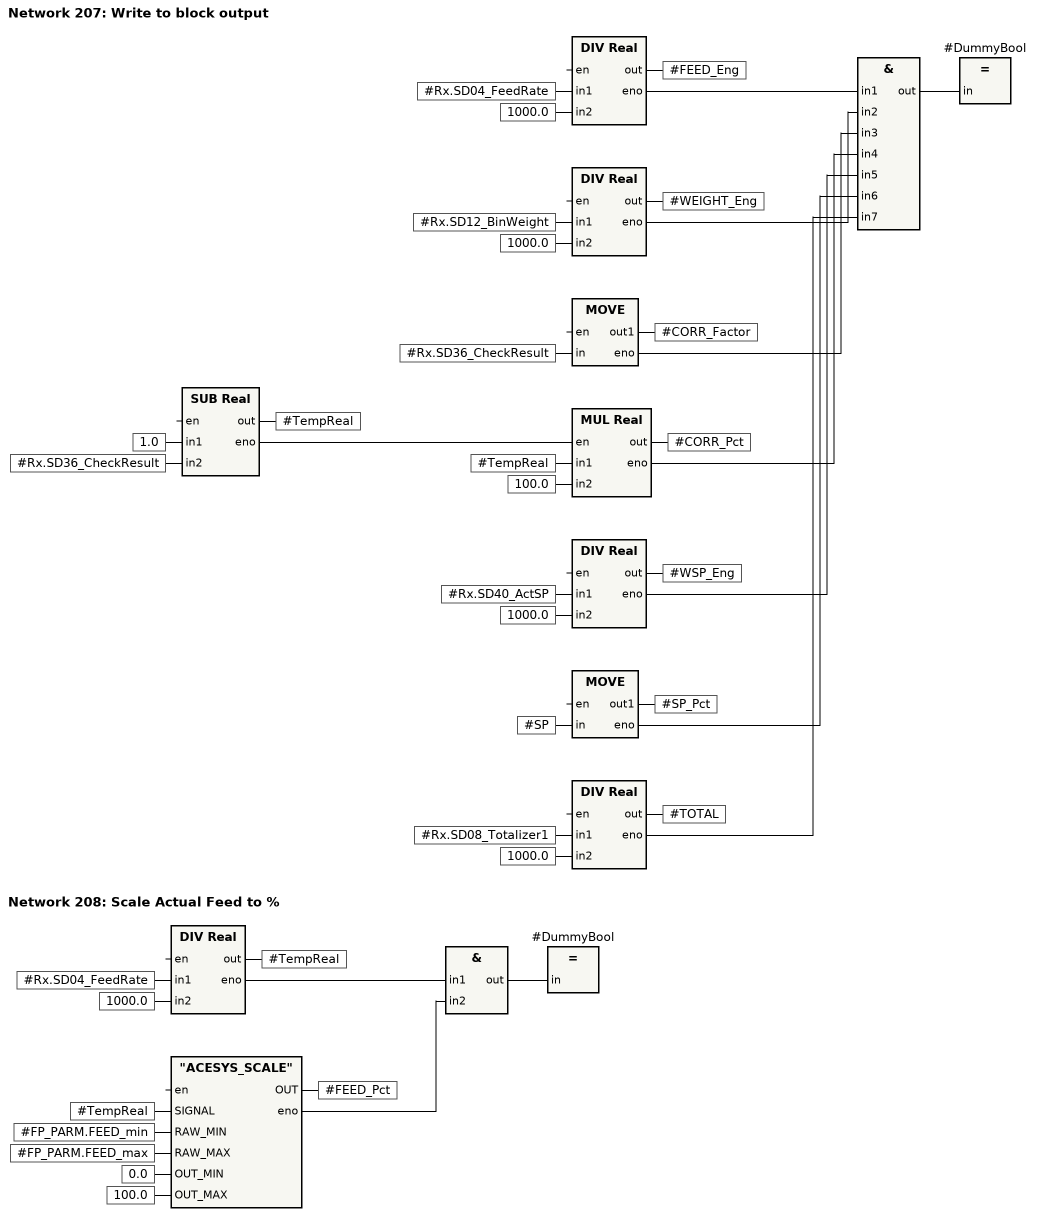
   // ENO of a box is taken as its EN; it also drops when the box reports an error
   #FEED_Eng := #Rx.SD04_FeedRate / 1000.0;
   #WEIGHT_Eng := #Rx.SD12_BinWeight / 1000.0;
   #CORR_Factor := #Rx.SD36_CheckResult;
   #TempReal := 1.0 - #Rx.SD36_CheckResult;
   #CORR_Pct := #TempReal * 100.0;
   #WSP_Eng := #Rx.SD40_ActSP / 1000.0;
   #SP_Pct := #SP;
   #TOTAL := #Rx.SD08_Totalizer1 / 1000.0;
   #DummyBool := TRUE;
END_REGION

REGION Network 208: Scale Actual Feed to %
   // ENO of a box is taken as its EN; it also drops when the box reports an error
   #TempReal := #Rx.SD04_FeedRate / 1000.0;
   "ACESYS_SCALE"(SIGNAL := #TempReal,
                  RAW_MIN := #FP_PARM.FEED_min,
                  RAW_MAX := #FP_PARM.FEED_max,
                  OUT_MIN := 0.0,
                  OUT_MAX := 100.0,
                  OUT => #FEED_Pct,
                  ENO => #_w1);
   #DummyBool := #_w1;
END_REGION

REGION Network 209: Scale Actual Setpoint to %
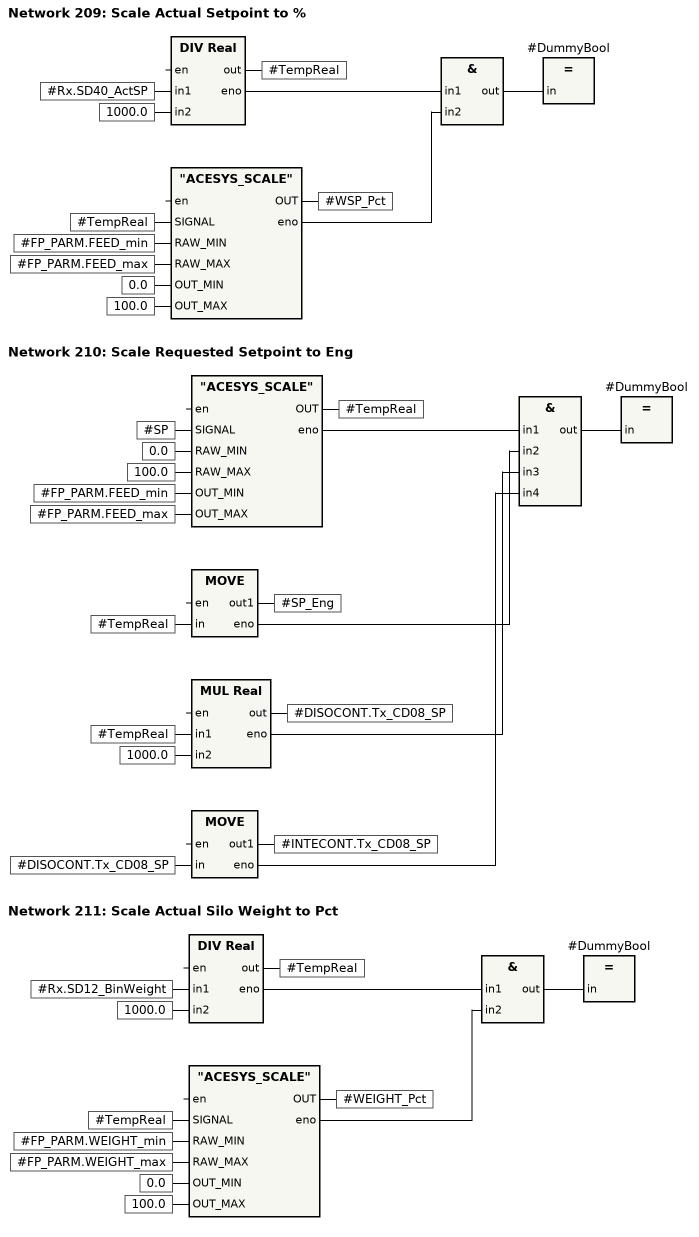
   // ENO of a box is taken as its EN; it also drops when the box reports an error
   #TempReal := #Rx.SD40_ActSP / 1000.0;
   "ACESYS_SCALE"(SIGNAL := #TempReal,
                  RAW_MIN := #FP_PARM.FEED_min,
                  RAW_MAX := #FP_PARM.FEED_max,
                  OUT_MIN := 0.0,
                  OUT_MAX := 100.0,
                  OUT => #WSP_Pct,
                  ENO => #_w1);
   #DummyBool := #_w1;
END_REGION

REGION Network 210: Scale Requested Setpoint to Eng
   // ENO of a box is taken as its EN; it also drops when the box reports an error
   "ACESYS_SCALE"(SIGNAL := #SP,
                  RAW_MIN := 0.0,
                  RAW_MAX := 100.0,
                  OUT_MIN := #FP_PARM.FEED_min,
                  OUT_MAX := #FP_PARM.FEED_max,
                  OUT => #TempReal,
                  ENO => #_w1);
   #SP_Eng := #TempReal;
   #DISOCONT.Tx_CD08_SP := #TempReal * 1000.0;
   #INTECONT.Tx_CD08_SP := #DISOCONT.Tx_CD08_SP;
   #DummyBool := #_w1;
END_REGION

REGION Network 211: Scale Actual Silo Weight to Pct
   // Build 002 - 27 March 2019 : Feed_Max flag in Outmax input is replaced with 100.0
   // ENO of a box is taken as its EN; it also drops when the box reports an error
   #TempReal := #Rx.SD12_BinWeight / 1000.0;
   "ACESYS_SCALE"(SIGNAL := #TempReal,
                  RAW_MIN := #FP_PARM.WEIGHT_min,
                  RAW_MAX := #FP_PARM.WEIGHT_max,
                  OUT_MIN := 0.0,
                  OUT_MAX := 100.0,
                  OUT => #WEIGHT_Pct,
                  ENO => #_w1);
   #DummyBool := #_w1;
END_REGION

REGION Network 212: Start On-Stream Calibation
   // Build 002 - 27 March 2019 : FSTOP flag is added in Reset condition
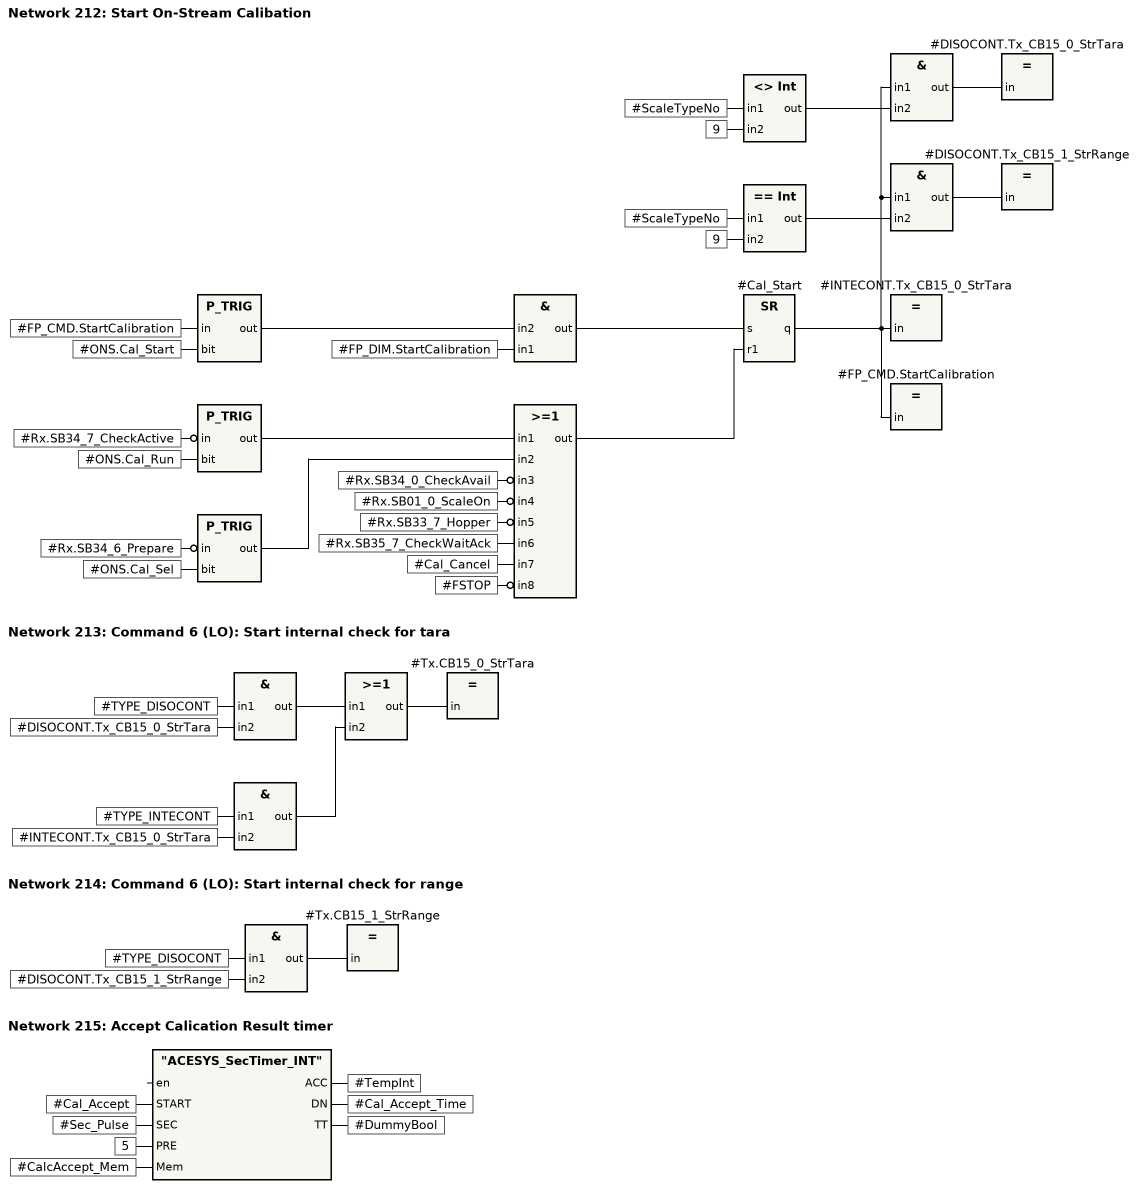
   #_w1 := #FP_CMD.StartCalibration AND NOT #ONS.Cal_Start;   // rising edge
   #ONS.Cal_Start := #FP_CMD.StartCalibration;
   #_w2 := NOT #Rx.SB34_7_CheckActive AND NOT #ONS.Cal_Run;   // rising edge
   #ONS.Cal_Run := NOT #Rx.SB34_7_CheckActive;
   #_w3 := NOT #Rx.SB34_6_Prepare AND NOT #ONS.Cal_Sel;   // rising edge
   #ONS.Cal_Sel := NOT #Rx.SB34_6_Prepare;
   IF #_w1 AND #FP_DIM.StartCalibration THEN
       #Cal_Start := TRUE;   // SR flip-flop
   END_IF;
   IF #_w2 OR #_w3 OR NOT #Rx.SB34_0_CheckAvail OR NOT #Rx.SB01_0_ScaleOn OR NOT #Rx.SB33_7_Hopper OR #Rx.SB35_7_CheckWaitAck OR #Cal_Cancel OR NOT #FSTOP THEN
       #Cal_Start := FALSE;
   END_IF;
   #DISOCONT.Tx_CB15_0_StrTara := #Cal_Start AND (#ScaleTypeNo <> 9);
   #DISOCONT.Tx_CB15_1_StrRange := #Cal_Start AND (#ScaleTypeNo = 9);
   #INTECONT.Tx_CB15_0_StrTara := #Cal_Start;
   #FP_CMD.StartCalibration := #Cal_Start;
END_REGION

REGION Network 213: Command 6 (LO): Start internal check for tara
   #Tx.CB15_0_StrTara := (#TYPE_DISOCONT AND #DISOCONT.Tx_CB15_0_StrTara) OR (#TYPE_INTECONT AND #INTECONT.Tx_CB15_0_StrTara);
END_REGION

REGION Network 214: Command 6 (LO): Start internal check for range
   #Tx.CB15_1_StrRange := #TYPE_DISOCONT AND #DISOCONT.Tx_CB15_1_StrRange;
END_REGION

REGION Network 215: Accept Calication Result timer
   // Timeout of the Acquire order
   "ACESYS_SecTimer_INT"(START := #Cal_Accept,
                         SEC := #Sec_Pulse,
                         PRE := 5,
                         Mem := #CalcAccept_Mem,
                         ACC => #TempInt,
                         DN => #Cal_Accept_Time,
                         TT => #DummyBool);
END_REGION

REGION Network 216: Accept Calibration Result
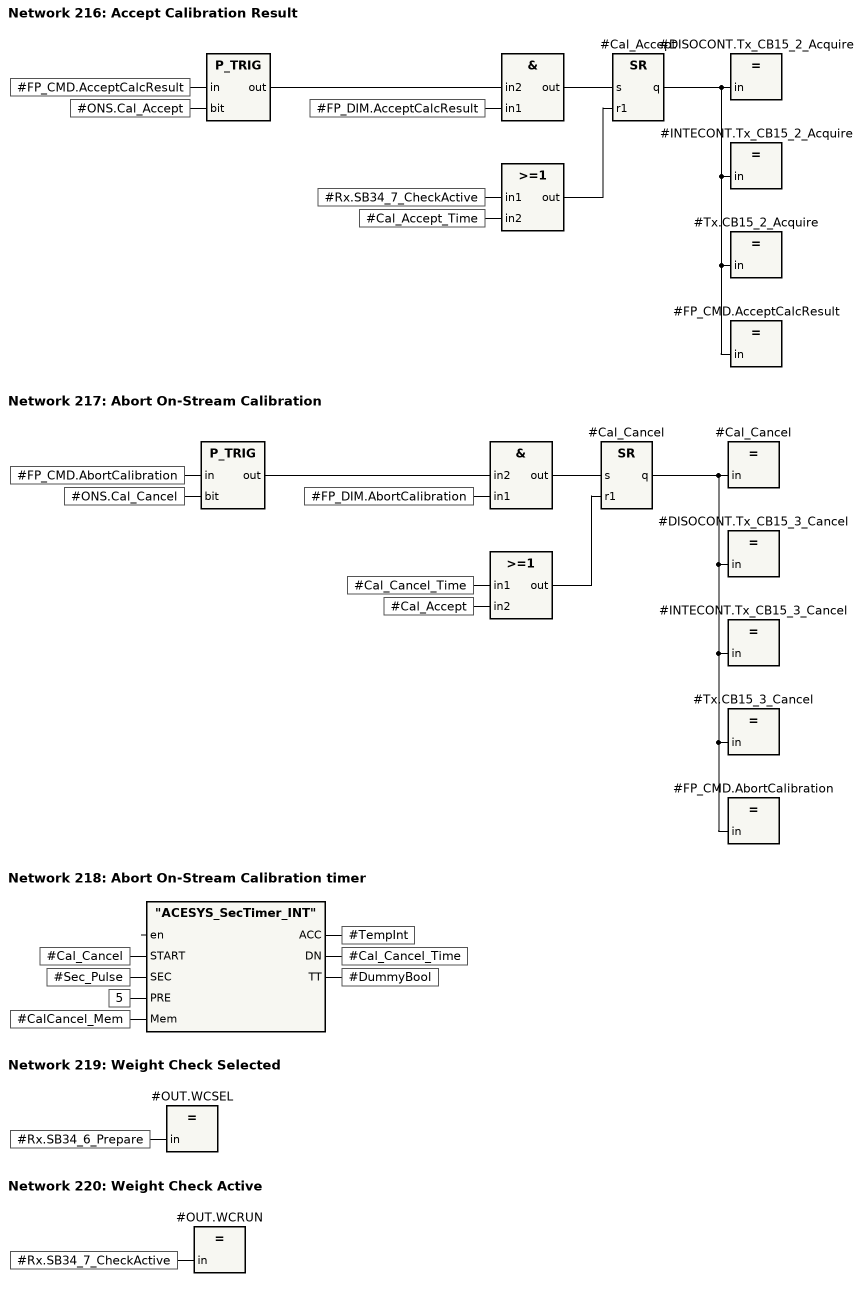
   #_w1 := #FP_CMD.AcceptCalcResult AND NOT #ONS.Cal_Accept;   // rising edge
   #ONS.Cal_Accept := #FP_CMD.AcceptCalcResult;
   IF #_w1 AND #FP_DIM.AcceptCalcResult THEN
       #Cal_Accept := TRUE;   // SR flip-flop
   END_IF;
   IF #Rx.SB34_7_CheckActive OR #Cal_Accept_Time THEN #Cal_Accept := FALSE; END_IF;
   #DISOCONT.Tx_CB15_2_Acquire := #Cal_Accept;
   #INTECONT.Tx_CB15_2_Acquire := #Cal_Accept;
   #Tx.CB15_2_Acquire := #Cal_Accept;
   #FP_CMD.AcceptCalcResult := #Cal_Accept;
END_REGION

REGION Network 217: Abort On-Stream Calibration
   #_w1 := #FP_CMD.AbortCalibration AND NOT #ONS.Cal_Cancel;   // rising edge
   #ONS.Cal_Cancel := #FP_CMD.AbortCalibration;
   IF #_w1 AND #FP_DIM.AbortCalibration THEN
       #Cal_Cancel := TRUE;   // SR flip-flop
   END_IF;
   IF #Cal_Cancel_Time OR #Cal_Accept THEN #Cal_Cancel := FALSE; END_IF;
   #_w2 := #Cal_Cancel;
   #Cal_Cancel := #Cal_Cancel;
   #DISOCONT.Tx_CB15_3_Cancel := #_w2;
   #INTECONT.Tx_CB15_3_Cancel := #_w2;
   #Tx.CB15_3_Cancel := #_w2;
   #FP_CMD.AbortCalibration := #_w2;
END_REGION

REGION Network 218: Abort On-Stream Calibration timer
   // Timeout of Abort order
   "ACESYS_SecTimer_INT"(START := #Cal_Cancel,
                         SEC := #Sec_Pulse,
                         PRE := 5,
                         Mem := #CalCancel_Mem,
                         ACC => #TempInt,
                         DN => #Cal_Cancel_Time,
                         TT => #DummyBool);
END_REGION

REGION Network 219: Weight Check Selected
   #OUT.WCSEL := #Rx.SB34_6_Prepare;
END_REGION

REGION Network 220: Weight Check Active
   #OUT.WCRUN := #Rx.SB34_7_CheckActive;
END_REGION

REGION Network 221: On-Stream Calibation block output status
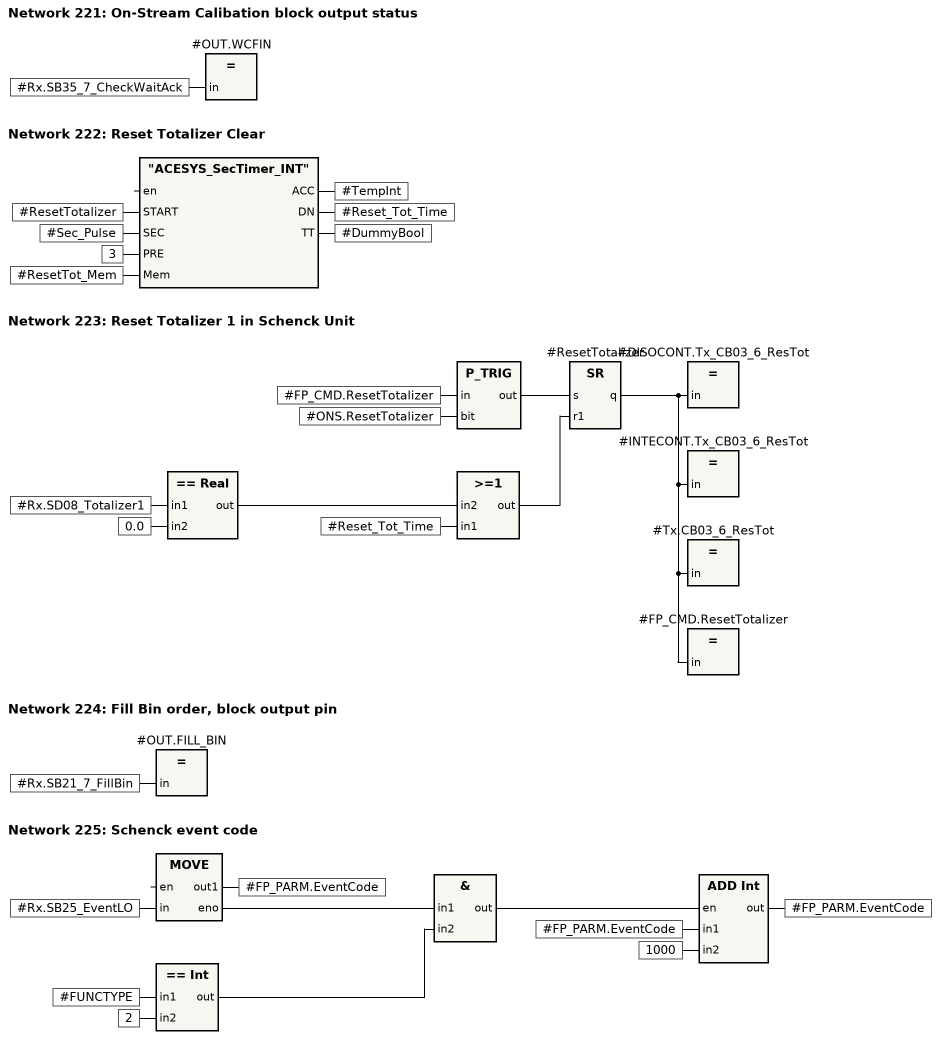
   #OUT.WCFIN := #Rx.SB35_7_CheckWaitAck;
END_REGION

REGION Network 222: Reset Totalizer Clear
   "ACESYS_SecTimer_INT"(START := #ResetTotalizer,
                         SEC := #Sec_Pulse,
                         PRE := 3,
                         Mem := #ResetTot_Mem,
                         ACC => #TempInt,
                         DN => #Reset_Tot_Time,
                         TT => #DummyBool);
END_REGION

REGION Network 223: Reset Totalizer 1 in Schenck Unit
   #_w1 := #FP_CMD.ResetTotalizer AND NOT #ONS.ResetTotalizer;   // rising edge
   #ONS.ResetTotalizer := #FP_CMD.ResetTotalizer;
   IF #_w1 THEN
       #ResetTotalizer := TRUE;   // SR flip-flop
   END_IF;
   IF (#Rx.SD08_Totalizer1 = 0.0) OR #Reset_Tot_Time THEN #ResetTotalizer := FALSE; END_IF;
   #DISOCONT.Tx_CB03_6_ResTot := #ResetTotalizer;
   #INTECONT.Tx_CB03_6_ResTot := #ResetTotalizer;
   #Tx.CB03_6_ResTot := #ResetTotalizer;
   #FP_CMD.ResetTotalizer := #ResetTotalizer;
END_REGION

REGION Network 224: Fill Bin order, block output pin
   #OUT.FILL_BIN := #Rx.SB21_7_FillBin;
END_REGION

REGION Network 225: Schenck event code
   // The byte Rx_SB25 represent the event group and number sendt from the Schenck 
   // equipment. 
   // 
   // With FUNCTYPE=1 (Disocont) the byte is moved direct to EventCode 
   // byte. 
   // 
   // With FUNCTYPE=2 (Intecont) the Rx_SB25 status is added 1000 before 
   // sending to EventCode byte. 
   // 
   // The EventCode number is translated to a text in the HMI faceplate.
   // ENO of a box is taken as its EN; it also drops when the box reports an error
   #FP_PARM.EventCode := #Rx.SB25_EventLO;
   IF #FUNCTYPE = 2 THEN #FP_PARM.EventCode := #FP_PARM.EventCode + 1000; END_IF;
END_REGION

REGION Network 226: Schenck Event Number
   // The event number is bit 0...3 of Rx_SB25 byte. The bits 4...7 are masked out 
   // and only the result of bit 0...3 are added "1" and moved to EventNo byte. 
   // 
   // The event numbers received from the Schenck Equipment are in the range 0...15, 
   // represention event no. 1...16.
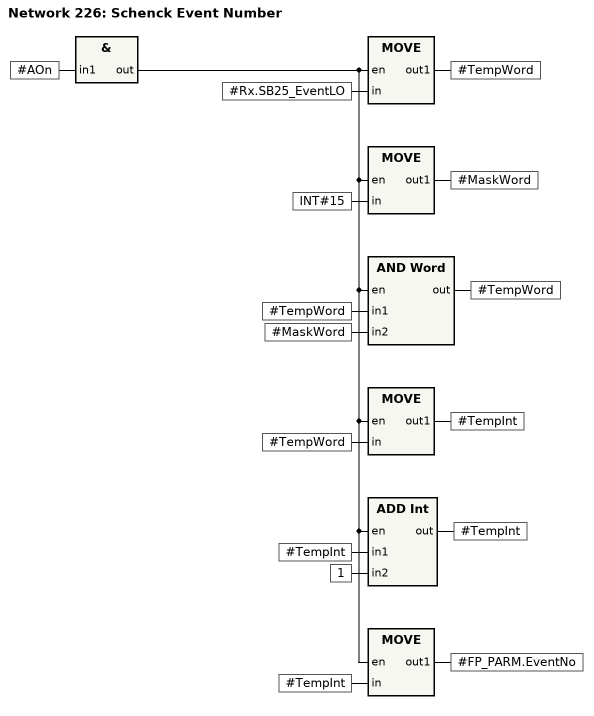
   IF #AOn THEN
       #TempWord := #Rx.SB25_EventLO;
       #MaskWord := INT#15;
       #TempWord := #TempWord AND #MaskWord;
       #TempInt := #TempWord;
       #TempInt := #TempInt + 1;
       #FP_PARM.EventNo := #TempInt;
   END_IF;
END_REGION

REGION Network 227: Schenck Event Group
   // The event number is bit 4..7 of Rx_SB25 byte. The bits 4...7 are shifted to 
   // bits 0...3 and the result is moved to the EventGrp byte.
   // 
   // With FUNCTYPE=2 (Intecont) the Rx_SB25 status is added 100 before sending 
   // to EventCode byte. 
   // The EventCode number is translated to text coding in the HMI faceplate.
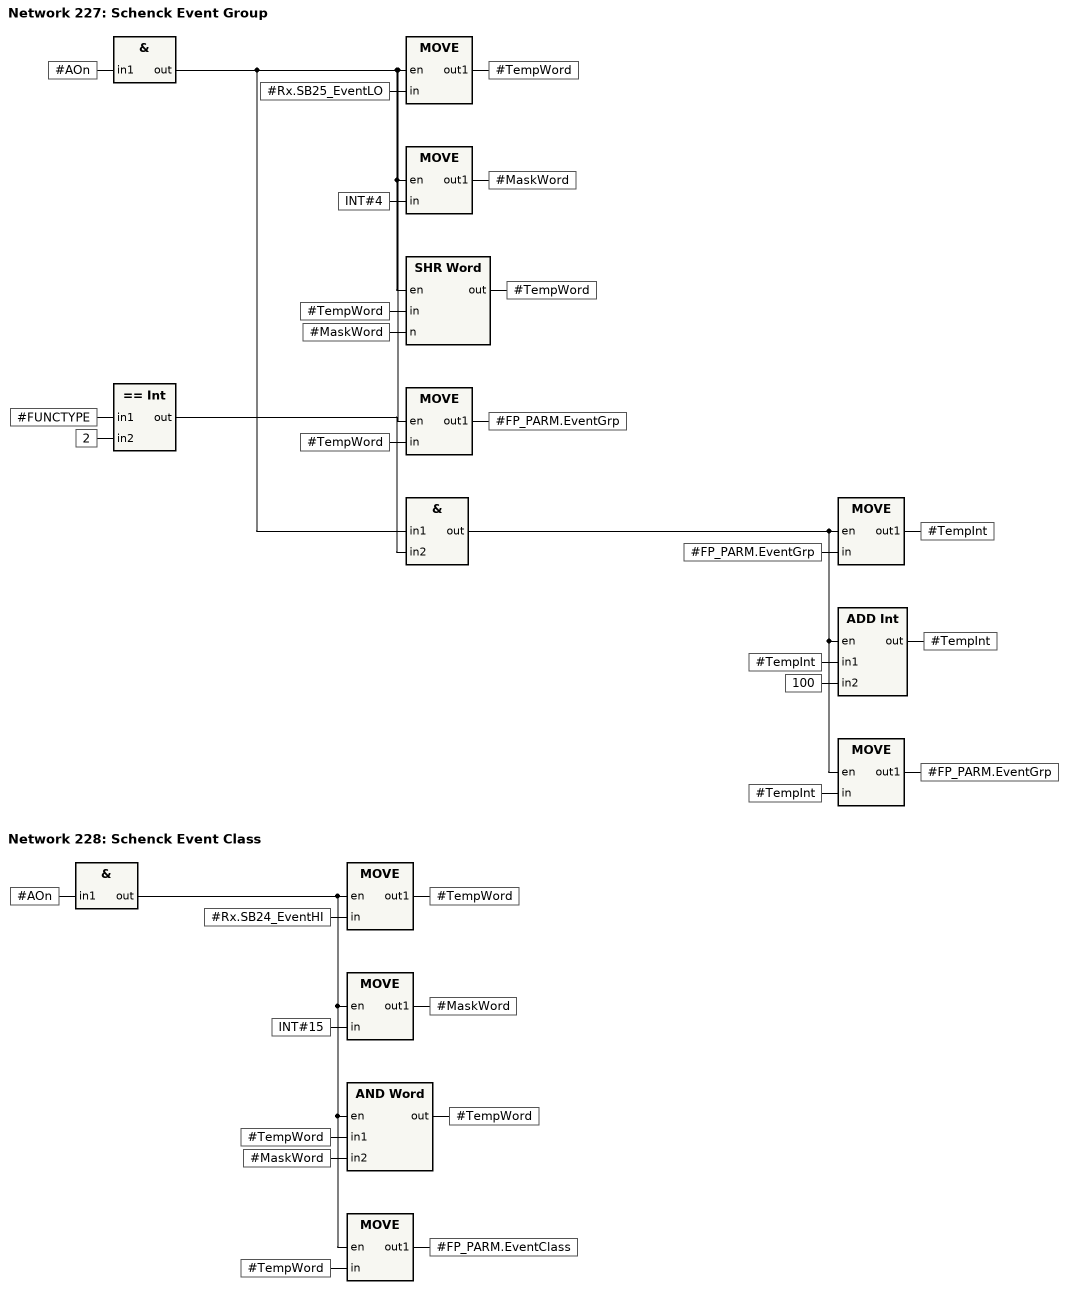
   IF #AOn THEN
       #TempWord := #Rx.SB25_EventLO;
       #MaskWord := INT#4;
       #TempWord := SHR(IN := #TempWord, N := #MaskWord);
       #FP_PARM.EventGrp := #TempWord;
   END_IF;
   IF #AOn AND (#FUNCTYPE = 2) THEN
       #TempInt := #FP_PARM.EventGrp;
       #TempInt := #TempInt + 100;
       #FP_PARM.EventGrp := #TempInt;
   END_IF;
END_REGION

REGION Network 228: Schenck Event Class
   // The event class is bit 0...3 of Rx_SB24 byte. The bits 4...7 are masked out and 
   // only the result of bit 0...3 are moved direct to EventClass byte. 
   // 
   // The EventClass number is translated to text coding in HMI.
   IF #AOn THEN
       #TempWord := #Rx.SB24_EventHI;
       #MaskWord := INT#15;
       #TempWord := #TempWord AND #MaskWord;
       #FP_PARM.EventClass := #TempWord;
   END_IF;
END_REGION

REGION Network 229: Schenck Event Acknowledge
   // The event acknowledge is bit 4...7 of Rx_SB24 byte. The bits 4...7 are shifted 
   // to bits 0...3 and the result is added "1" and moved to the EventAck byte. 
   // 
   // The value received from the Schenck Equipment is: 0=Unacknowledged and 
   // 1=Acknowledged. This is changed to: 1=Unacknowledged and 2=Acknowledged.
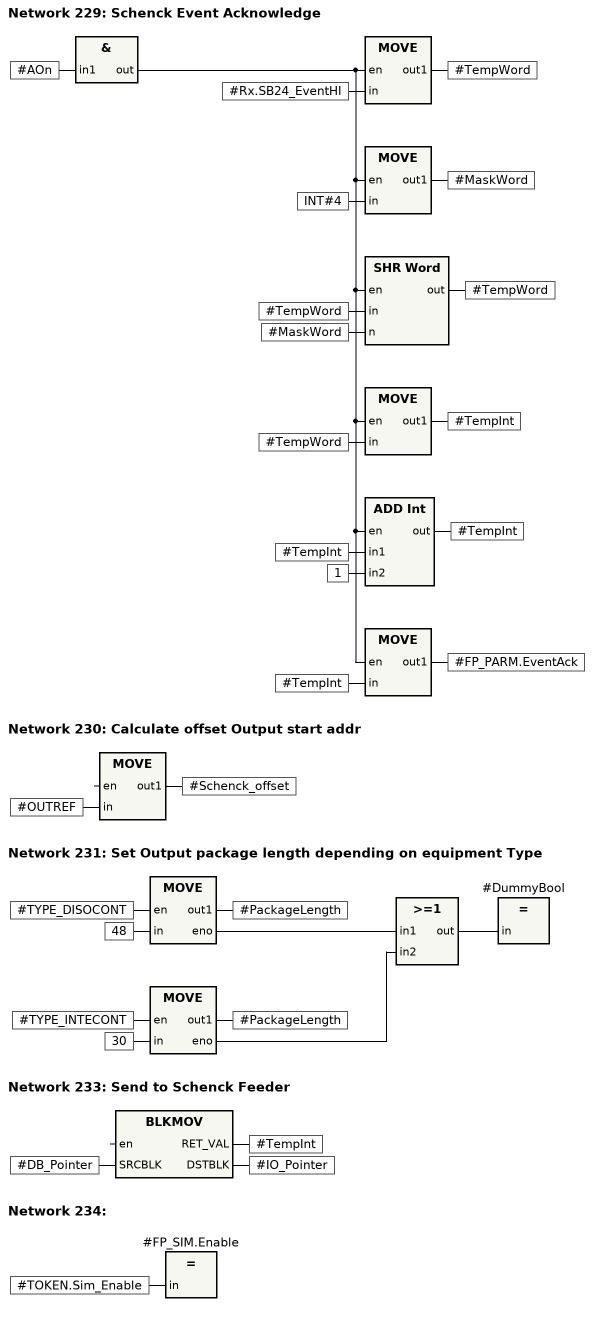
   IF #AOn THEN
       #TempWord := #Rx.SB24_EventHI;
       #MaskWord := INT#4;
       #TempWord := SHR(IN := #TempWord, N := #MaskWord);
       #TempInt := #TempWord;
       #TempInt := #TempInt + 1;
       #FP_PARM.EventAck := #TempInt;
   END_IF;
END_REGION

REGION Network 230: Calculate offset Output start addr
   // Hardware Address
   #Schenck_offset := #OUTREF;
END_REGION

REGION Network 231: Set Output package length depending on equipment Type
   // ENO of a box is taken as its EN; it also drops when the box reports an error
   IF #TYPE_DISOCONT THEN #PackageLength := 48; END_IF;
   IF #TYPE_INTECONT THEN #PackageLength := 30; END_IF;
   #DummyBool := #TYPE_DISOCONT OR #TYPE_INTECONT;
END_REGION

REGION Network 232 (STL): Target Pointers Sending Output Data
         LAR1;  // Make AR1 pointer to Unit Output
         L     16#10;  // ANY Syntax ID
         T     LB[AR1, P#0.0];  // ..Store Byte 0
         L     16#02;  // Data Type = Byte
         T     LB[AR1, P#1.0];  // ..Store Byte 1
         L     #PackageLength;  // Load Packed length
         T     LW[AR1, P#2.0];  // ..Store byte 2/3
         L     0;  // used with DB else "0"
         T     LW[AR1, P#4.0];  // ..Store byte 4/5
         L     #Schenck_offset;  // Source offset (Variable for Node's)
         SLD   3;  // with offset
         OD    16#8200_0000;  // Output Area (I/O) Code (S7)
         T     LD[AR1, P#6.0];  // ..Store byte 6/7/8/9
         LAR1;  // Make AR1 pointer to calling local stack Unit Output data
         L     16#10;  // ANY Syntax ID
         T     LB[AR1, P#0.0];  // ..Store Byte 0
         L     16#02;  // Data Type = Byte
         T     LB[AR1, P#1.0];  // ..Store Byte 1
         L     #PackageLength;  // Load Packed length
         T     LW[AR1, P#2.0];  // ..Store byte 2/3
         L     0;  // used with DB use No. else "0"
         T     LW[AR1, P#4.0];  // ..Store byte 4/5
         L     #FUNCTYPE;  // Load FuncType
         L     1;  // 1=DISOCONT
         <>I;
         JC    INTE;  // If not = 1 jump to INTECONT
         L;  // Load source offset DISOCONT
         JU    DONE;
   INTE: L;  // Load source offset INTECONT
   DONE: T     D[AR1, P#6.0];  // ..Store byte 6/7/8/9
         L     16#87;  // 87=Local Stack area
         T     B[AR1, P#6.0];  // ..Store byte 6
END_REGION

REGION Network 233: Send to Schenck Feeder
   #TempInt := BLKMOV(SRCBLK := #DB_Pointer, DSTBLK => #IO_Pointer);
END_REGION

REGION Network 234
   #FP_SIM.Enable := #TOKEN.Sim_Enable;
END_REGION

REGION Network 235: Set Simulation Enabled and calibation simulation
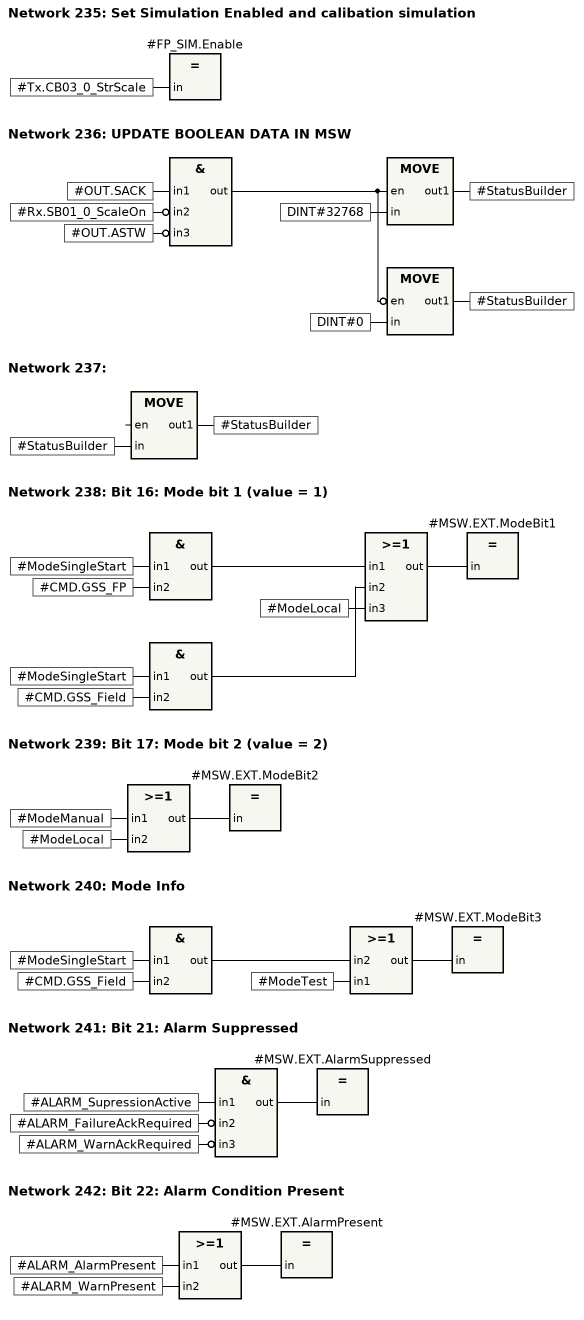
   #FP_SIM.Enable := #Tx.CB03_0_StrScale;
END_REGION

REGION Network 236: UPDATE BOOLEAN DATA IN MSW
   #_w1 := #OUT.SACK AND NOT #Rx.SB01_0_ScaleOn AND NOT #OUT.ASTW;
   IF #_w1 THEN #StatusBuilder := DINT#32768; END_IF;
   IF NOT #_w1 THEN #StatusBuilder := DINT#0; END_IF;
END_REGION

REGION Network 237
   #StatusBuilder := #StatusBuilder;
END_REGION

REGION Network 238: Bit 16: Mode bit 1 (value = 1)
   #MSW.EXT.ModeBit1 := (#ModeSingleStart AND #CMD.GSS_FP) OR (#ModeSingleStart AND #CMD.GSS_Field) OR #ModeLocal;
END_REGION

REGION Network 239: Bit 17: Mode bit 2 (value = 2)
   #MSW.EXT.ModeBit2 := #ModeManual OR #ModeLocal;
END_REGION

REGION Network 240: Mode Info
   #MSW.EXT.ModeBit3 := (#ModeSingleStart AND #CMD.GSS_Field) OR #ModeTest;
END_REGION

REGION Network 241: Bit 21: Alarm Suppressed
   #MSW.EXT.AlarmSuppressed := #ALARM_SupressionActive AND NOT #ALARM_FailureAckRequired AND NOT #ALARM_WarnAckRequired;
END_REGION

REGION Network 242: Bit 22: Alarm Condition Present
   #MSW.EXT.AlarmPresent := #ALARM_AlarmPresent OR #ALARM_WarnPresent;
END_REGION

REGION Network 243: Bit 23: Alarm Failure Present or Unacknowledged
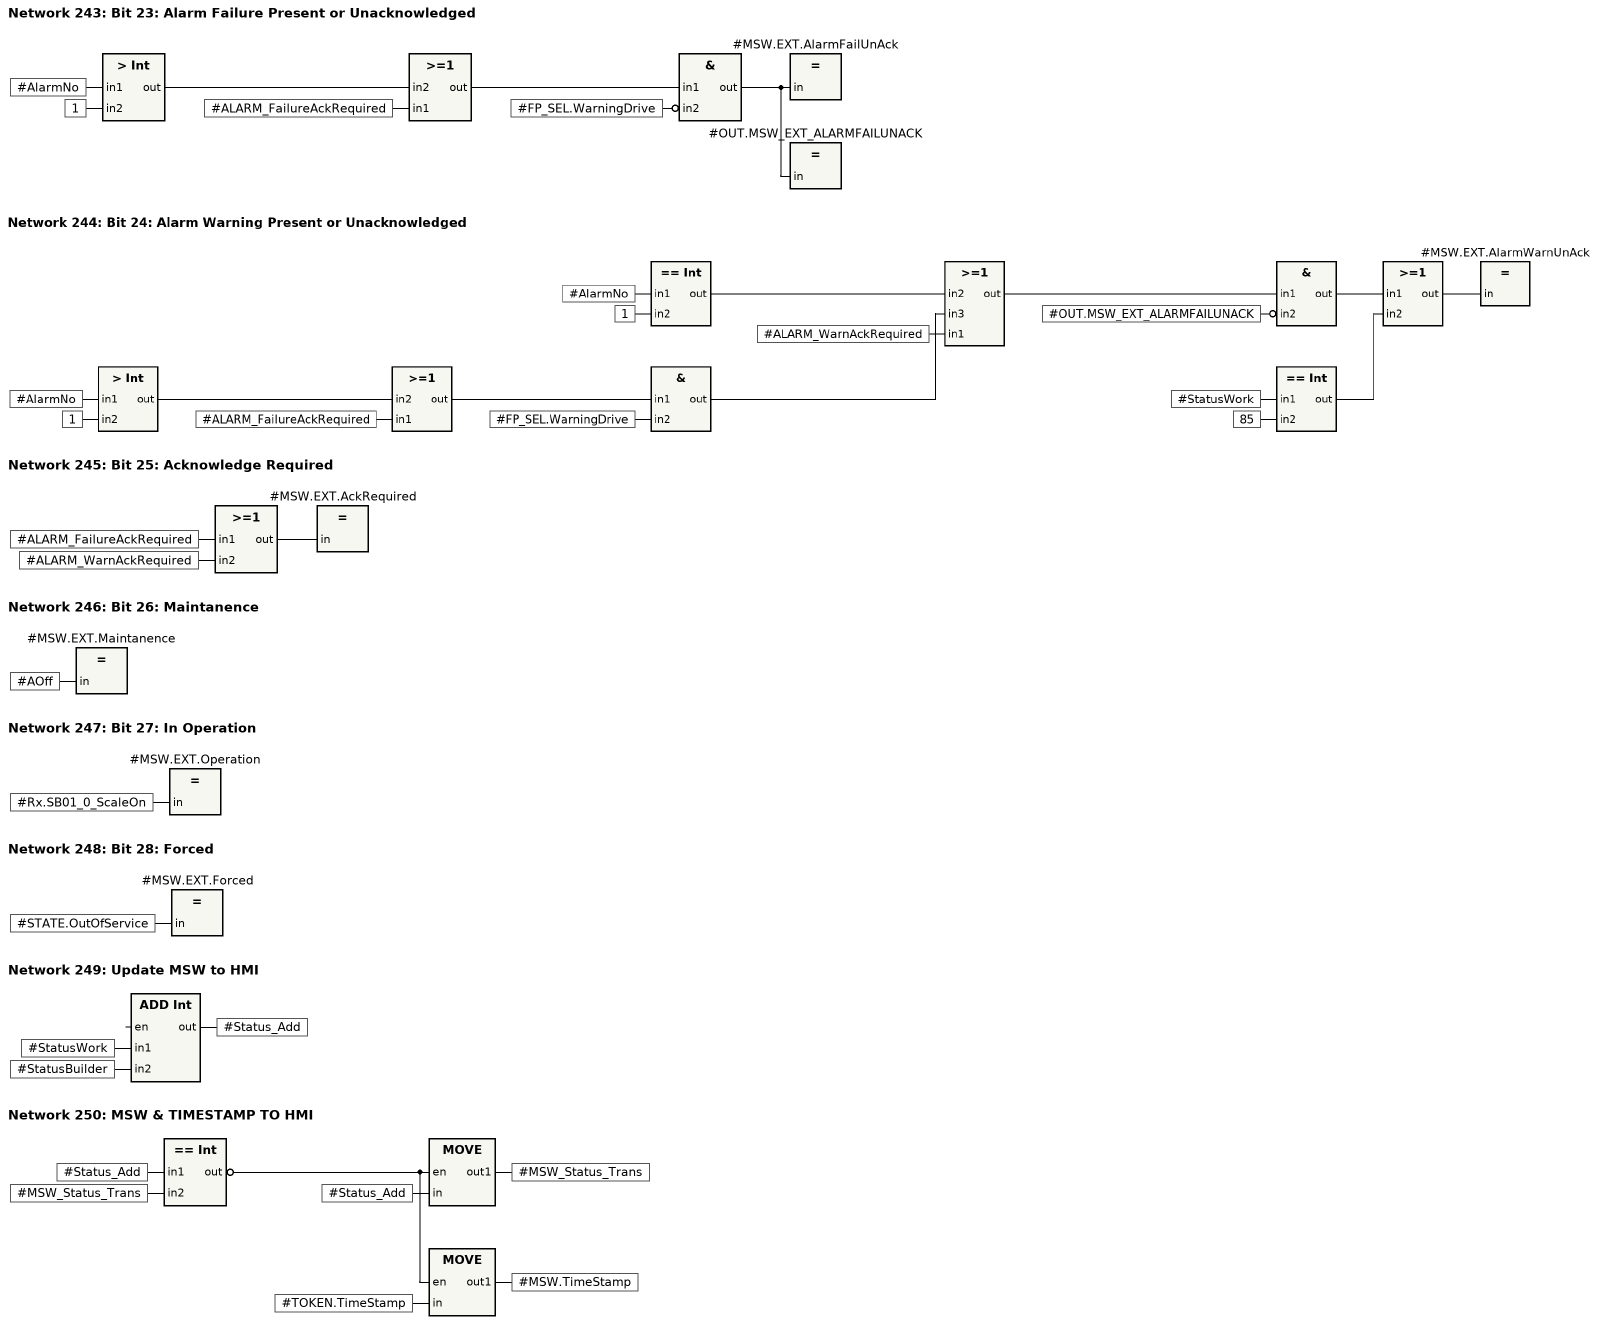
   #MSW.EXT.AlarmFailUnAck := ((#AlarmNo > 1) OR #ALARM_FailureAckRequired) AND NOT #FP_SEL.WarningDrive;
   #OUT.MSW_EXT_ALARMFAILUNACK := #MSW.EXT.AlarmFailUnAck;
END_REGION

REGION Network 244: Bit 24: Alarm Warning Present or Unacknowledged
   #MSW.EXT.AlarmWarnUnAck := (((#AlarmNo = 1) OR (((#AlarmNo > 1) OR #ALARM_FailureAckRequired) AND #FP_SEL.WarningDrive) OR #ALARM_WarnAckRequired) AND NOT #OUT.MSW_EXT_ALARMFAILUNACK) OR (#StatusWork = 85);
END_REGION

REGION Network 245: Bit 25: Acknowledge Required
   #MSW.EXT.AckRequired := #ALARM_FailureAckRequired OR #ALARM_WarnAckRequired;
END_REGION

REGION Network 246: Bit 26: Maintanence
   #MSW.EXT.Maintanence := #AOff;
END_REGION

REGION Network 247: Bit 27: In Operation
   #MSW.EXT.Operation := #Rx.SB01_0_ScaleOn;
END_REGION

REGION Network 248: Bit 28: Forced
   // Build 002 - 27 March 2019 : new network : bit 28 - Forced with State.OutofService
   #MSW.EXT.Forced := #STATE.OutOfService;
END_REGION

REGION Network 249: Update MSW to HMI
   #Status_Add := #StatusWork + #StatusBuilder;
END_REGION

REGION Network 250: MSW & TIMESTAMP TO HMI
   #_w1 := NOT (#Status_Add = #MSW_Status_Trans);
   IF #_w1 THEN
       #MSW_Status_Trans := #Status_Add;
       #MSW.TimeStamp := #TOKEN.TimeStamp;
   END_IF;
END_REGION

REGION Network 251: MSW Transfer to Actual
